(* IEC 61131-3 sources: open-ot-experiments/st/iec61131/src, 5 files *)

(* ---- openot_message.st ---- *)
FUNCTION_BLOCK OPENOT_EncodeMinimalMessage
VAR_INPUT
    SourceId : UDINT;
    RunId : ULINT;
    Seq : ULINT;
    SourceTime : ULINT;
    MessageTemplateId : UDINT;
END_VAR
VAR_OUTPUT
    Buffer : OPENOT_BYTE_BUFFER;
    Length : UINT;
END_VAR
VAR
    Pos : UINT;
    Crc : DWORD;
END_VAR

Pos := OPENOT_WriteHeader(
    TotalLength := UINT#52,
    Flags := UINT#16#0008,
    SourceTime := SourceTime,
    RunId := RunId,
    Seq := Seq,
    SourceId := SourceId,
    EventTypeId := UDINT#16#0003,
    Buffer := Buffer);

Pos := OPENOT_WriteSlotHeader(
    Offset := Pos,
    Key := UINT#16#0014,
    TypeTag := BYTE#16#05,
    PayloadLength := BYTE#4,
    Buffer := Buffer);
Pos := OPENOT_WriteU32LE(Offset := Pos, Value := MessageTemplateId, Buffer := Buffer);

Crc := OPENOT_Crc32c(Data := Buffer, Length := Pos);
Pos := OPENOT_WriteDWordLE(Offset := Pos, Value := Crc, Buffer := Buffer);
Length := Pos;
END_FUNCTION_BLOCK

(* ---- openot_producer.st ---- *)
TYPE
    OPENOT_SOURCE_ENTRY : STRUCT
        Used : BOOL;
        SourceId : UDINT;
        NextSeq : ULINT;
    END_STRUCT;

    OPENOT_SOURCE_USED_TABLE : ARRAY[0..15] OF BOOL;
    OPENOT_SOURCE_ID_TABLE : ARRAY[0..15] OF UDINT;
    OPENOT_SOURCE_NEXT_SEQ_TABLE : ARRAY[0..15] OF ULINT;
    OPENOT_SCAN_RECORD_BUFFER : ARRAY[0..1023] OF BYTE;
    OPENOT_SCAN_RECORD_UINT_TABLE : ARRAY[0..16] OF UINT;

    OPENOT_REAL_VALUE_STATE : STRUCT
        Used : BOOL;
        ValueId : UDINT;
        HasLast : BOOL;
        LastValue : REAL;
    END_STRUCT;

    OPENOT_INT_VALUE_STATE : STRUCT
        Used : BOOL;
        ValueId : UDINT;
        HasLast : BOOL;
        LastValue : DINT;
    END_STRUCT;

    OPENOT_STATE_MACHINE_STATE : STRUCT
        Used : BOOL;
        StateMachineId : UDINT;
        HasLast : BOOL;
        LastState : UINT;
    END_STRUCT;

    OPENOT_CONDITION_STATE : STRUCT
        Used : BOOL;
        ConditionId : UDINT;
        HasLast : BOOL;
        LastActive : BOOL;
    END_STRUCT;

    OPENOT_EMISSION_ENTRY : STRUCT
        EventTypeId : UDINT;
        RunId : ULINT;
        SourceId : UDINT;
        Seq : ULINT;
    END_STRUCT;

    OPENOT_EMISSION_LOG : ARRAY[0..31] OF OPENOT_EMISSION_ENTRY;
END_TYPE

FUNCTION OPENOT_AppendScanRecord : BOOL
VAR_INPUT
    Record : OPENOT_BYTE_BUFFER;
    Length : UINT;
END_VAR
VAR_IN_OUT
    ScanRecords : OPENOT_SCAN_RECORD_BUFFER;
    ScanRecordOffsets : OPENOT_SCAN_RECORD_UINT_TABLE;
    ScanRecordLengths : OPENOT_SCAN_RECORD_UINT_TABLE;
    ScanWritePos : UINT;
    ScanRecordCount : UINT;
END_VAR
VAR
    CopyIndex : UINT;
    DestIndex : UINT;
END_VAR

IF (Length = UINT#0) OR (Length > UINT#256) OR (ScanRecordCount > UINT#16) OR ((ScanWritePos + Length) > UINT#1024) THEN
    OPENOT_AppendScanRecord := FALSE;
ELSE
    ScanRecordOffsets[ScanRecordCount] := ScanWritePos;
    ScanRecordLengths[ScanRecordCount] := Length;

    FOR CopyIndex := UINT#0 TO Length - UINT#1 DO
        DestIndex := ScanWritePos + CopyIndex;
        ScanRecords[DestIndex] := Record[CopyIndex];
    END_FOR;

    ScanWritePos := ScanWritePos + Length;
    ScanRecordCount := ScanRecordCount + UINT#1;
    OPENOT_AppendScanRecord := TRUE;
END_IF;
END_FUNCTION

FUNCTION OPENOT_ResetScanRecordList : BOOL
VAR_IN_OUT
    ScanRecordOffsets : OPENOT_SCAN_RECORD_UINT_TABLE;
    ScanRecordLengths : OPENOT_SCAN_RECORD_UINT_TABLE;
    ScanWritePos : UINT;
    ScanRecordCount : UINT;
END_VAR
VAR
    Index : UINT;
END_VAR

ScanRecordCount := UINT#0;
ScanWritePos := UINT#0;
FOR Index := UINT#0 TO UINT#16 DO
    ScanRecordOffsets[Index] := UINT#0;
    ScanRecordLengths[Index] := UINT#0;
END_FOR;

OPENOT_ResetScanRecordList := TRUE;
END_FUNCTION

FUNCTION OPENOT_NextSourceTime : ULINT
VAR_INPUT
    UseSourceTimeInput : BOOL;
    SourceTimeInput : ULINT;
END_VAR
VAR_IN_OUT
    StateSourceTime : ULINT;
END_VAR

IF UseSourceTimeInput THEN
    OPENOT_NextSourceTime := SourceTimeInput;
ELSE
    OPENOT_NextSourceTime := StateSourceTime;
    StateSourceTime := StateSourceTime + ULINT#1;
END_IF;
END_FUNCTION

FUNCTION_BLOCK OPENOT_Producer
VAR_INPUT
    Execute : BOOL;
    Op : UINT;
    SourceId : UDINT;
    Checkpoint : BOOL;
    DefHashOld : OPENOT_HASH8;
    DefHashNew : OPENOT_HASH8;
    TransitionEpochId : ULINT;
    UseSourceTimeInput : BOOL;
    SourceTimeInput : ULINT;
    StageRecord : OPENOT_BYTE_BUFFER;
    StageLength : UINT;
    StageSeq : ULINT;
    StageEventTypeId : UDINT;
    ResetScanRecords : BOOL;
    AccumulateScanRecords : BOOL;
    ValueId : UDINT;
    ValueReal : REAL;
    ValueInt : DINT;
    DeadbandReal : REAL;
    HasQuality : BOOL;
    Quality : UINT;
    StateMachineId : UDINT;
    Category : UINT;
    PreviousState : UINT;
    NewState : UINT;
    ConditionId : UDINT;
    ConditionClass : UINT;
    Severity : UINT;
    ConditionActive : BOOL;
    MessageTemplateId : UDINT;
END_VAR
VAR_OUTPUT
    AssignedSeq : ULINT;
    ProducedCount : ULINT;
    Error : BOOL;
    SourceTableFull : BOOL;
    Done : BOOL;
    CheckpointDone : BOOL;
    SourceCount : UINT;
    SourceUsed : OPENOT_SOURCE_USED_TABLE;
    SourceIds : OPENOT_SOURCE_ID_TABLE;
    SourceNextSeqs : OPENOT_SOURCE_NEXT_SEQ_TABLE;
    Ring : OPENOT_RING256_BUFFER;
    HeadAbs : ULINT;
    OldestAbs : ULINT;
    LostCount : ULINT;
    LastStartAbs : ULINT;
    LastEndAbs : ULINT;
    LossRanges : OPENOT_PRODUCER_LOSS_RANGES;
    LossRangeCount : UINT;
    LossRangeOverflow : BOOL;
    RingError : BOOL;
    RunId : ULINT;
    SourceTime : ULINT;
    SystemSeq : ULINT;
    EpochId : ULINT;
    EpochFirstAbs : ULINT;
    DefinitionHash : OPENOT_HASH8;
    PrevDefinitionHash : OPENOT_HASH8;
    TransitionOpen : BOOL;
    DefinitionChangedEmitted : BOOL;
    Emissions : OPENOT_EMISSION_LOG;
    EmissionCount : UINT;
    PublishedRecordCount : ULINT;
    ScanRecords : OPENOT_SCAN_RECORD_BUFFER;
    ScanRecordOffsets : OPENOT_SCAN_RECORD_UINT_TABLE;
    ScanRecordLengths : OPENOT_SCAN_RECORD_UINT_TABLE;
    ScanRecordCount : UINT;
END_VAR
VAR
    Sources : ARRAY[0..15] OF OPENOT_SOURCE_ENTRY;
    RealValueStates : ARRAY[0..15] OF OPENOT_REAL_VALUE_STATE;
    IntValueStates : ARRAY[0..15] OF OPENOT_INT_VALUE_STATE;
    StateMachineStates : ARRAY[0..15] OF OPENOT_STATE_MACHINE_STATE;
    ConditionStates : ARRAY[0..15] OF OPENOT_CONDITION_STATE;
    RingProducer : OPENOT_Ring256Producer;
    Encoder : OPENOT_EncodeMinimalMessage;
    ValueRealEncoder : OPENOT_EncodeValueChangedReal;
    ValueIntEncoder : OPENOT_EncodeValueChangedInt;
    StateTransitionEncoder : OPENOT_EncodeStateTransition;
    ConditionEncoder : OPENOT_EncodeCondition;
    HighWaterEncoder : OPENOT_EncodeSourceHighWater;
    StoppedEncoder : OPENOT_EncodeLoggerStopped;
    StartedEncoder : OPENOT_EncodeLoggerStarted;
    DefinitionEncoder : OPENOT_EncodeDefinitionChanged;
    Index : UINT;
    ByteIndex : UINT;
    LossIndex : UINT;
    EntryIndex : UINT;
    Found : BOOL;
    FreeFound : BOOL;
    Initialized : BOOL;
    PreviousExecute : BOOL;
    ExecuteEdge : BOOL;
    StateRunId : ULINT;
    StateSourceTime : ULINT;
    StateSystemSeq : ULINT;
    StateEpochId : ULINT;
    StateEpochFirstAbs : ULINT;
    StateDefinitionHash : OPENOT_HASH8;
    StatePrevDefinitionHash : OPENOT_HASH8;
    StatePublishedRecordCount : ULINT;
    PendingDefHashOld : OPENOT_HASH8;
    PendingDefHashNew : OPENOT_HASH8;
    PendingEpochId : ULINT;
    PendingOpen : BOOL;
    PendingDefChangedEmitted : BOOL;
    EmitSeq : ULINT;
    EmitSourceTime : ULINT;
    SourceLoopActive : BOOL;
    HasLastSourceId : BOOL;
    LastSourceId : UDINT;
    NextSourceId : UDINT;
    SelectedIndex : UINT;
    StateIndex : UINT;
    StateFound : BOOL;
    StateFreeFound : BOOL;
    ActiveSourceId : UDINT;
    ShouldEmit : BOOL;
    DeltaReal : REAL;
    CandidateFound : BOOL;
    ScanWritePos : UINT;
    AppendOk : BOOL;
    ResetOk : BOOL;
    ConditionEventTypeId : UDINT;
END_VAR

IF NOT Initialized THEN
    StateRunId := ULINT#1;
    StateSourceTime := ULINT#1780000000000000000;
    StateSystemSeq := ULINT#0;
    StateEpochId := ULINT#1;
    StateEpochFirstAbs := ULINT#0;
    StatePublishedRecordCount := ULINT#0;
    Initialized := TRUE;
END_IF;

Done := FALSE;
Error := FALSE;
SourceTableFull := FALSE;
AssignedSeq := ULINT#0;
ProducedCount := ULINT#0;
CheckpointDone := FALSE;
ExecuteEdge := Execute AND (NOT PreviousExecute);

IF ResetScanRecords THEN
    ResetOk := OPENOT_ResetScanRecordList(
        ScanRecordOffsets := ScanRecordOffsets,
        ScanRecordLengths := ScanRecordLengths,
        ScanWritePos := ScanWritePos,
        ScanRecordCount := ScanRecordCount);
END_IF;

IF ExecuteEdge THEN
    IF (NOT AccumulateScanRecords) AND (Op <> UINT#6) AND (Op <> UINT#7) AND (Op <> UINT#8) AND (Op <> UINT#9) THEN
        ResetOk := OPENOT_ResetScanRecordList(
            ScanRecordOffsets := ScanRecordOffsets,
            ScanRecordLengths := ScanRecordLengths,
            ScanWritePos := ScanWritePos,
            ScanRecordCount := ScanRecordCount);
    END_IF;

    IF Checkpoint THEN
        IF PendingOpen THEN
            Error := TRUE;
        ELSIF SourceId = UDINT#0 THEN
            Error := TRUE;
        ELSE
            Found := FALSE;
            EntryIndex := UINT#0;

            FOR Index := UINT#0 TO UINT#15 DO
                IF Sources[Index].Used AND (Sources[Index].SourceId = SourceId) THEN
                    IF NOT Found THEN
                        EntryIndex := Index;
                        Found := TRUE;
                    END_IF;
                END_IF;
            END_FOR;

            IF NOT Found THEN
                Error := TRUE;
            ELSE
                ProducedCount := Sources[EntryIndex].NextSeq;
                EmitSourceTime := OPENOT_NextSourceTime(
                    UseSourceTimeInput := UseSourceTimeInput,
                    SourceTimeInput := SourceTimeInput,
                    StateSourceTime := StateSourceTime);
                HighWaterEncoder(
                    SourceId := SourceId,
                    RunId := StateRunId,
                    ProducedCount := ProducedCount,
                    SourceTime := EmitSourceTime);
                RingProducer(
                    Execute := TRUE,
                    Record := HighWaterEncoder.Buffer,
                    Length := HighWaterEncoder.Length,
                    RunId := StateRunId,
                    SourceId := SourceId,
                    Seq := ProducedCount);

                IF RingProducer.Done AND (NOT RingProducer.Error) THEN
                    AppendOk := OPENOT_AppendScanRecord(
                        Record := HighWaterEncoder.Buffer,
                        Length := HighWaterEncoder.Length,
                        ScanRecords := ScanRecords,
                        ScanRecordOffsets := ScanRecordOffsets,
                        ScanRecordLengths := ScanRecordLengths,
                        ScanWritePos := ScanWritePos,
                        ScanRecordCount := ScanRecordCount);
                    IF AppendOk THEN
                        Sources[EntryIndex].NextSeq := ProducedCount + ULINT#1;
                        StatePublishedRecordCount := StatePublishedRecordCount + ULINT#1;
                        IF EmissionCount < UINT#32 THEN
                            Emissions[EmissionCount].EventTypeId := UDINT#16#80000108;
                            Emissions[EmissionCount].RunId := StateRunId;
                            Emissions[EmissionCount].SourceId := SourceId;
                            Emissions[EmissionCount].Seq := ProducedCount;
                            EmissionCount := EmissionCount + UINT#1;
                        END_IF;
                        Done := TRUE;
                        CheckpointDone := TRUE;
                    ELSE
                        Error := TRUE;
                    END_IF;
                ELSE
                    Error := TRUE;
                END_IF;
            END_IF;
        END_IF;
    ELSIF Op = UINT#0 THEN
        IF PendingOpen THEN
            Error := TRUE;
        ELSIF SourceId = UDINT#0 THEN
            Error := TRUE;
        ELSE
            Found := FALSE;
            FreeFound := FALSE;
            EntryIndex := UINT#0;

            FOR Index := UINT#0 TO UINT#15 DO
                IF Sources[Index].Used AND (Sources[Index].SourceId = SourceId) THEN
                    IF NOT Found THEN
                        EntryIndex := Index;
                        Found := TRUE;
                    END_IF;
                END_IF;
            END_FOR;

            IF NOT Found THEN
                FOR Index := UINT#0 TO UINT#15 DO
                    IF (NOT Sources[Index].Used) AND (NOT FreeFound) THEN
                        EntryIndex := Index;
                        FreeFound := TRUE;
                    END_IF;
                END_FOR;

                IF FreeFound THEN
                    Sources[EntryIndex].Used := TRUE;
                    Sources[EntryIndex].SourceId := SourceId;
                    Sources[EntryIndex].NextSeq := ULINT#0;
                ELSE
                    SourceTableFull := TRUE;
                    Error := TRUE;
                END_IF;
            END_IF;

            IF NOT Error THEN
                AssignedSeq := Sources[EntryIndex].NextSeq;
                Sources[EntryIndex].NextSeq := Sources[EntryIndex].NextSeq + ULINT#1;
                EmitSourceTime := OPENOT_NextSourceTime(
                    UseSourceTimeInput := UseSourceTimeInput,
                    SourceTimeInput := SourceTimeInput,
                    StateSourceTime := StateSourceTime);

                Encoder(
                    SourceId := SourceId,
                    RunId := StateRunId,
                    Seq := AssignedSeq,
                    SourceTime := EmitSourceTime,
                    MessageTemplateId := MessageTemplateId);
                RingProducer(
                    Execute := TRUE,
                    Record := Encoder.Buffer,
                    Length := Encoder.Length,
                    RunId := StateRunId,
                    SourceId := SourceId,
                    Seq := AssignedSeq);

                IF RingProducer.Done AND (NOT RingProducer.Error) THEN
                    AppendOk := OPENOT_AppendScanRecord(
                        Record := Encoder.Buffer,
                        Length := Encoder.Length,
                        ScanRecords := ScanRecords,
                        ScanRecordOffsets := ScanRecordOffsets,
                        ScanRecordLengths := ScanRecordLengths,
                        ScanWritePos := ScanWritePos,
                        ScanRecordCount := ScanRecordCount);
                    IF AppendOk THEN
                        StatePublishedRecordCount := StatePublishedRecordCount + ULINT#1;
                        IF EmissionCount < UINT#32 THEN
                            Emissions[EmissionCount].EventTypeId := UDINT#16#0003;
                            Emissions[EmissionCount].RunId := StateRunId;
                            Emissions[EmissionCount].SourceId := SourceId;
                            Emissions[EmissionCount].Seq := AssignedSeq;
                            EmissionCount := EmissionCount + UINT#1;
                        END_IF;
                        Done := TRUE;
                    ELSE
                        Error := TRUE;
                    END_IF;
                ELSE
                    Error := TRUE;
                END_IF;
            END_IF;
        END_IF;
    ELSIF Op = UINT#5 THEN
        IF PendingOpen THEN
            Error := TRUE;
        ELSIF SourceId = UDINT#0 THEN
            Error := TRUE;
        ELSIF (StageLength = UINT#0) OR (StageLength > UINT#256) THEN
            Error := TRUE;
        ELSE
            Found := FALSE;
            FreeFound := FALSE;
            EntryIndex := UINT#0;

            FOR Index := UINT#0 TO UINT#15 DO
                IF Sources[Index].Used AND (Sources[Index].SourceId = SourceId) THEN
                    IF NOT Found THEN
                        EntryIndex := Index;
                        Found := TRUE;
                    END_IF;
                END_IF;
            END_FOR;

            IF NOT Found THEN
                FOR Index := UINT#0 TO UINT#15 DO
                    IF (NOT Sources[Index].Used) AND (NOT FreeFound) THEN
                        EntryIndex := Index;
                        FreeFound := TRUE;
                    END_IF;
                END_FOR;

                IF FreeFound THEN
                    Sources[EntryIndex].Used := TRUE;
                    Sources[EntryIndex].SourceId := SourceId;
                    Sources[EntryIndex].NextSeq := ULINT#0;
                ELSE
                    SourceTableFull := TRUE;
                    Error := TRUE;
                END_IF;
            END_IF;

            IF NOT Error THEN
                IF StageSeq <> Sources[EntryIndex].NextSeq THEN
                    Error := TRUE;
                ELSE
                    RingProducer(
                        Execute := TRUE,
                        Record := StageRecord,
                        Length := StageLength,
                        RunId := StateRunId,
                        SourceId := SourceId,
                        Seq := StageSeq);

                    IF RingProducer.Done AND (NOT RingProducer.Error) THEN
                        AppendOk := OPENOT_AppendScanRecord(
                            Record := StageRecord,
                            Length := StageLength,
                            ScanRecords := ScanRecords,
                            ScanRecordOffsets := ScanRecordOffsets,
                            ScanRecordLengths := ScanRecordLengths,
                            ScanWritePos := ScanWritePos,
                            ScanRecordCount := ScanRecordCount);
                        IF AppendOk THEN
                            AssignedSeq := StageSeq;
                            Sources[EntryIndex].NextSeq := StageSeq + ULINT#1;
                            StatePublishedRecordCount := StatePublishedRecordCount + ULINT#1;
                            IF EmissionCount < UINT#32 THEN
                                Emissions[EmissionCount].EventTypeId := StageEventTypeId;
                                Emissions[EmissionCount].RunId := StateRunId;
                                Emissions[EmissionCount].SourceId := SourceId;
                                Emissions[EmissionCount].Seq := StageSeq;
                                EmissionCount := EmissionCount + UINT#1;
                            END_IF;
                            Done := TRUE;
                        ELSE
                            Error := TRUE;
                        END_IF;
                    ELSE
                        Error := TRUE;
                    END_IF;
                END_IF;
            END_IF;
        END_IF;
    ELSIF (Op = UINT#6) OR (Op = UINT#7) OR (Op = UINT#8) THEN
        ActiveSourceId := SourceId;
        IF ActiveSourceId = UDINT#0 THEN
            ActiveSourceId := UDINT#1;
        END_IF;

        StateFound := FALSE;
        StateFreeFound := FALSE;
        StateIndex := UINT#0;
        ShouldEmit := FALSE;

        IF Op = UINT#6 THEN
            IF ValueId = UDINT#0 THEN
                Error := TRUE;
            ELSE
                FOR Index := UINT#0 TO UINT#15 DO
                    IF RealValueStates[Index].Used AND (RealValueStates[Index].ValueId = ValueId) THEN
                        IF NOT StateFound THEN
                            StateIndex := Index;
                            StateFound := TRUE;
                        END_IF;
                    ELSIF (NOT StateFound) AND (NOT RealValueStates[Index].Used) AND (NOT StateFreeFound) THEN
                        StateIndex := Index;
                        StateFreeFound := TRUE;
                    END_IF;
                END_FOR;

                IF StateFound THEN
                    IF RealValueStates[StateIndex].HasLast THEN
                        DeltaReal := ValueReal - RealValueStates[StateIndex].LastValue;
                        IF DeltaReal < REAL#0.0 THEN
                            DeltaReal := REAL#0.0 - DeltaReal;
                        END_IF;
                        ShouldEmit := DeltaReal > DeadbandReal;
                    ELSE
                        ShouldEmit := TRUE;
                    END_IF;
                ELSIF StateFreeFound THEN
                    RealValueStates[StateIndex].Used := TRUE;
                    RealValueStates[StateIndex].ValueId := ValueId;
                    RealValueStates[StateIndex].HasLast := FALSE;
                    ShouldEmit := TRUE;
                ELSE
                    Error := TRUE;
                END_IF;
            END_IF;
        ELSIF Op = UINT#7 THEN
            IF ValueId = UDINT#0 THEN
                Error := TRUE;
            ELSE
                FOR Index := UINT#0 TO UINT#15 DO
                    IF IntValueStates[Index].Used AND (IntValueStates[Index].ValueId = ValueId) THEN
                        IF NOT StateFound THEN
                            StateIndex := Index;
                            StateFound := TRUE;
                        END_IF;
                    ELSIF (NOT StateFound) AND (NOT IntValueStates[Index].Used) AND (NOT StateFreeFound) THEN
                        StateIndex := Index;
                        StateFreeFound := TRUE;
                    END_IF;
                END_FOR;

                IF StateFound THEN
                    IF IntValueStates[StateIndex].HasLast THEN
                        ShouldEmit := ValueInt <> IntValueStates[StateIndex].LastValue;
                    ELSE
                        ShouldEmit := TRUE;
                    END_IF;
                ELSIF StateFreeFound THEN
                    IntValueStates[StateIndex].Used := TRUE;
                    IntValueStates[StateIndex].ValueId := ValueId;
                    IntValueStates[StateIndex].HasLast := FALSE;
                    ShouldEmit := TRUE;
                ELSE
                    Error := TRUE;
                END_IF;
            END_IF;
        ELSE
            IF StateMachineId = UDINT#0 THEN
                Error := TRUE;
            ELSE
                FOR Index := UINT#0 TO UINT#15 DO
                    IF StateMachineStates[Index].Used AND (StateMachineStates[Index].StateMachineId = StateMachineId) THEN
                        IF NOT StateFound THEN
                            StateIndex := Index;
                            StateFound := TRUE;
                        END_IF;
                    ELSIF (NOT StateFound) AND (NOT StateMachineStates[Index].Used) AND (NOT StateFreeFound) THEN
                        StateIndex := Index;
                        StateFreeFound := TRUE;
                    END_IF;
                END_FOR;

                IF PreviousState <> NewState THEN
                    IF StateFound THEN
                        ShouldEmit := (NOT StateMachineStates[StateIndex].HasLast) OR (StateMachineStates[StateIndex].LastState <> NewState);
                    ELSIF StateFreeFound THEN
                        StateMachineStates[StateIndex].Used := TRUE;
                        StateMachineStates[StateIndex].StateMachineId := StateMachineId;
                        StateMachineStates[StateIndex].HasLast := FALSE;
                        ShouldEmit := TRUE;
                    ELSE
                        Error := TRUE;
                    END_IF;
                ELSE
                    ShouldEmit := FALSE;
                END_IF;
            END_IF;
        END_IF;

        IF (NOT Error) AND (NOT ShouldEmit) THEN
            Done := TRUE;
        ELSIF NOT Error THEN
            Found := FALSE;
            FreeFound := FALSE;
            EntryIndex := UINT#0;

            FOR Index := UINT#0 TO UINT#15 DO
                IF Sources[Index].Used AND (Sources[Index].SourceId = ActiveSourceId) THEN
                    IF NOT Found THEN
                        EntryIndex := Index;
                        Found := TRUE;
                    END_IF;
                END_IF;
            END_FOR;

            IF NOT Found THEN
                FOR Index := UINT#0 TO UINT#15 DO
                    IF (NOT Sources[Index].Used) AND (NOT FreeFound) THEN
                        EntryIndex := Index;
                        FreeFound := TRUE;
                    END_IF;
                END_FOR;

                IF FreeFound THEN
                    Sources[EntryIndex].Used := TRUE;
                    Sources[EntryIndex].SourceId := ActiveSourceId;
                    Sources[EntryIndex].NextSeq := ULINT#0;
                ELSE
                    SourceTableFull := TRUE;
                    Error := TRUE;
                END_IF;
            END_IF;

            IF NOT Error THEN
                AssignedSeq := Sources[EntryIndex].NextSeq;
                EmitSourceTime := OPENOT_NextSourceTime(
                    UseSourceTimeInput := UseSourceTimeInput,
                    SourceTimeInput := SourceTimeInput,
                    StateSourceTime := StateSourceTime);

                IF Op = UINT#6 THEN
                    ValueRealEncoder(
                        SourceId := ActiveSourceId,
                        RunId := StateRunId,
                        Seq := AssignedSeq,
                        SourceTime := EmitSourceTime,
                        ValueId := ValueId,
                        NewValue := ValueReal,
                        HasPrevious := RealValueStates[StateIndex].HasLast,
                        PreviousValue := RealValueStates[StateIndex].LastValue,
                        HasQuality := HasQuality,
                        Quality := Quality);
                    RingProducer(
                        Execute := TRUE,
                        Record := ValueRealEncoder.Buffer,
                        Length := ValueRealEncoder.Length,
                        RunId := StateRunId,
                        SourceId := ActiveSourceId,
                        Seq := AssignedSeq);

                    IF RingProducer.Done AND (NOT RingProducer.Error) THEN
                        AppendOk := OPENOT_AppendScanRecord(
                            Record := ValueRealEncoder.Buffer,
                            Length := ValueRealEncoder.Length,
                            ScanRecords := ScanRecords,
                            ScanRecordOffsets := ScanRecordOffsets,
                            ScanRecordLengths := ScanRecordLengths,
                            ScanWritePos := ScanWritePos,
                            ScanRecordCount := ScanRecordCount);
                    ELSE
                        AppendOk := FALSE;
                    END_IF;
                ELSIF Op = UINT#7 THEN
                    ValueIntEncoder(
                        SourceId := ActiveSourceId,
                        RunId := StateRunId,
                        Seq := AssignedSeq,
                        SourceTime := EmitSourceTime,
                        ValueId := ValueId,
                        NewValue := ValueInt,
                        HasPrevious := IntValueStates[StateIndex].HasLast,
                        PreviousValue := IntValueStates[StateIndex].LastValue,
                        HasQuality := HasQuality,
                        Quality := Quality);
                    RingProducer(
                        Execute := TRUE,
                        Record := ValueIntEncoder.Buffer,
                        Length := ValueIntEncoder.Length,
                        RunId := StateRunId,
                        SourceId := ActiveSourceId,
                        Seq := AssignedSeq);

                    IF RingProducer.Done AND (NOT RingProducer.Error) THEN
                        AppendOk := OPENOT_AppendScanRecord(
                            Record := ValueIntEncoder.Buffer,
                            Length := ValueIntEncoder.Length,
                            ScanRecords := ScanRecords,
                            ScanRecordOffsets := ScanRecordOffsets,
                            ScanRecordLengths := ScanRecordLengths,
                            ScanWritePos := ScanWritePos,
                            ScanRecordCount := ScanRecordCount);
                    ELSE
                        AppendOk := FALSE;
                    END_IF;
                ELSE
                    StateTransitionEncoder(
                        SourceId := ActiveSourceId,
                        RunId := StateRunId,
                        Seq := AssignedSeq,
                        SourceTime := EmitSourceTime,
                        StateMachineId := StateMachineId,
                        Category := Category,
                        PreviousState := PreviousState,
                        NewState := NewState);
                    RingProducer(
                        Execute := TRUE,
                        Record := StateTransitionEncoder.Buffer,
                        Length := StateTransitionEncoder.Length,
                        RunId := StateRunId,
                        SourceId := ActiveSourceId,
                        Seq := AssignedSeq);

                    IF RingProducer.Done AND (NOT RingProducer.Error) THEN
                        AppendOk := OPENOT_AppendScanRecord(
                            Record := StateTransitionEncoder.Buffer,
                            Length := StateTransitionEncoder.Length,
                            ScanRecords := ScanRecords,
                            ScanRecordOffsets := ScanRecordOffsets,
                            ScanRecordLengths := ScanRecordLengths,
                            ScanWritePos := ScanWritePos,
                            ScanRecordCount := ScanRecordCount);
                    ELSE
                        AppendOk := FALSE;
                    END_IF;
                END_IF;

                IF AppendOk THEN
                    Sources[EntryIndex].NextSeq := AssignedSeq + ULINT#1;
                    StatePublishedRecordCount := StatePublishedRecordCount + ULINT#1;
                    IF EmissionCount < UINT#32 THEN
                        IF Op = UINT#8 THEN
                            Emissions[EmissionCount].EventTypeId := UDINT#16#0001;
                        ELSE
                            Emissions[EmissionCount].EventTypeId := UDINT#16#0002;
                        END_IF;
                        Emissions[EmissionCount].RunId := StateRunId;
                        Emissions[EmissionCount].SourceId := ActiveSourceId;
                        Emissions[EmissionCount].Seq := AssignedSeq;
                        EmissionCount := EmissionCount + UINT#1;
                    END_IF;

                    IF Op = UINT#6 THEN
                        RealValueStates[StateIndex].HasLast := TRUE;
                        RealValueStates[StateIndex].LastValue := ValueReal;
                    ELSIF Op = UINT#7 THEN
                        IntValueStates[StateIndex].HasLast := TRUE;
                        IntValueStates[StateIndex].LastValue := ValueInt;
                    ELSE
                        StateMachineStates[StateIndex].HasLast := TRUE;
                        StateMachineStates[StateIndex].LastState := NewState;
                    END_IF;
                    Done := TRUE;
                ELSE
                    Error := TRUE;
                END_IF;
            END_IF;
        END_IF;
    ELSIF Op = UINT#9 THEN
        ActiveSourceId := SourceId;
        IF ActiveSourceId = UDINT#0 THEN
            ActiveSourceId := UDINT#1;
        END_IF;

        StateFound := FALSE;
        StateFreeFound := FALSE;
        StateIndex := UINT#0;
        ShouldEmit := FALSE;

        IF ConditionId = UDINT#0 THEN
            Error := TRUE;
        ELSE
            FOR Index := UINT#0 TO UINT#15 DO
                IF ConditionStates[Index].Used AND (ConditionStates[Index].ConditionId = ConditionId) THEN
                    IF NOT StateFound THEN
                        StateIndex := Index;
                        StateFound := TRUE;
                    END_IF;
                ELSIF (NOT StateFound) AND (NOT ConditionStates[Index].Used) AND (NOT StateFreeFound) THEN
                    StateIndex := Index;
                    StateFreeFound := TRUE;
                END_IF;
            END_FOR;

            IF StateFound THEN
                IF ConditionStates[StateIndex].HasLast THEN
                    ShouldEmit := ConditionStates[StateIndex].LastActive <> ConditionActive;
                ELSE
                    ShouldEmit := ConditionActive;
                END_IF;
            ELSIF StateFreeFound THEN
                ConditionStates[StateIndex].Used := TRUE;
                ConditionStates[StateIndex].ConditionId := ConditionId;
                ConditionStates[StateIndex].HasLast := FALSE;
                ShouldEmit := ConditionActive;
            ELSE
                Error := TRUE;
            END_IF;
        END_IF;

        IF (NOT Error) AND (NOT ShouldEmit) THEN
            IF StateFound OR StateFreeFound THEN
                ConditionStates[StateIndex].HasLast := TRUE;
                ConditionStates[StateIndex].LastActive := ConditionActive;
            END_IF;
            Done := TRUE;
        ELSIF NOT Error THEN
            Found := FALSE;
            FreeFound := FALSE;
            EntryIndex := UINT#0;

            FOR Index := UINT#0 TO UINT#15 DO
                IF Sources[Index].Used AND (Sources[Index].SourceId = ActiveSourceId) THEN
                    IF NOT Found THEN
                        EntryIndex := Index;
                        Found := TRUE;
                    END_IF;
                END_IF;
            END_FOR;

            IF NOT Found THEN
                FOR Index := UINT#0 TO UINT#15 DO
                    IF (NOT Sources[Index].Used) AND (NOT FreeFound) THEN
                        EntryIndex := Index;
                        FreeFound := TRUE;
                    END_IF;
                END_FOR;

                IF FreeFound THEN
                    Sources[EntryIndex].Used := TRUE;
                    Sources[EntryIndex].SourceId := ActiveSourceId;
                    Sources[EntryIndex].NextSeq := ULINT#0;
                ELSE
                    SourceTableFull := TRUE;
                    Error := TRUE;
                END_IF;
            END_IF;

            IF NOT Error THEN
                AssignedSeq := Sources[EntryIndex].NextSeq;
                EmitSourceTime := OPENOT_NextSourceTime(
                    UseSourceTimeInput := UseSourceTimeInput,
                    SourceTimeInput := SourceTimeInput,
                    StateSourceTime := StateSourceTime);
                IF ConditionActive THEN
                    ConditionEventTypeId := UDINT#16#0200;
                ELSE
                    ConditionEventTypeId := UDINT#16#0201;
                END_IF;

                ConditionEncoder(
                    SourceId := ActiveSourceId,
                    RunId := StateRunId,
                    Seq := AssignedSeq,
                    SourceTime := EmitSourceTime,
                    EventTypeId := ConditionEventTypeId,
                    ConditionId := ConditionId,
                    ConditionClass := ConditionClass,
                    Severity := Severity);
                RingProducer(
                    Execute := TRUE,
                    Record := ConditionEncoder.Buffer,
                    Length := ConditionEncoder.Length,
                    RunId := StateRunId,
                    SourceId := ActiveSourceId,
                    Seq := AssignedSeq);

                IF RingProducer.Done AND (NOT RingProducer.Error) THEN
                    AppendOk := OPENOT_AppendScanRecord(
                        Record := ConditionEncoder.Buffer,
                        Length := ConditionEncoder.Length,
                        ScanRecords := ScanRecords,
                        ScanRecordOffsets := ScanRecordOffsets,
                        ScanRecordLengths := ScanRecordLengths,
                        ScanWritePos := ScanWritePos,
                        ScanRecordCount := ScanRecordCount);
                ELSE
                    AppendOk := FALSE;
                END_IF;

                IF AppendOk THEN
                    Sources[EntryIndex].NextSeq := AssignedSeq + ULINT#1;
                    StatePublishedRecordCount := StatePublishedRecordCount + ULINT#1;
                    IF EmissionCount < UINT#32 THEN
                        Emissions[EmissionCount].EventTypeId := ConditionEventTypeId;
                        Emissions[EmissionCount].RunId := StateRunId;
                        Emissions[EmissionCount].SourceId := ActiveSourceId;
                        Emissions[EmissionCount].Seq := AssignedSeq;
                        EmissionCount := EmissionCount + UINT#1;
                    END_IF;
                    ConditionStates[StateIndex].HasLast := TRUE;
                    ConditionStates[StateIndex].LastActive := ConditionActive;
                    Done := TRUE;
                ELSE
                    Error := TRUE;
                END_IF;
            END_IF;
        END_IF;
    ELSIF Op = UINT#1 THEN
        IF PendingOpen THEN
            Error := TRUE;
        ELSE
            EmitSeq := StateSystemSeq;
            StateSystemSeq := StateSystemSeq + ULINT#1;
            EmitSourceTime := OPENOT_NextSourceTime(
                UseSourceTimeInput := UseSourceTimeInput,
                SourceTimeInput := SourceTimeInput,
                StateSourceTime := StateSourceTime);
            StoppedEncoder(RunId := StateRunId, Seq := EmitSeq, SourceTime := EmitSourceTime);
            RingProducer(
                Execute := TRUE,
                Record := StoppedEncoder.Buffer,
                Length := StoppedEncoder.Length,
                RunId := StateRunId,
                SourceId := UDINT#0,
                Seq := EmitSeq);

            IF RingProducer.Done AND (NOT RingProducer.Error) THEN
                AppendOk := OPENOT_AppendScanRecord(
                    Record := StoppedEncoder.Buffer,
                    Length := StoppedEncoder.Length,
                    ScanRecords := ScanRecords,
                    ScanRecordOffsets := ScanRecordOffsets,
                    ScanRecordLengths := ScanRecordLengths,
                    ScanWritePos := ScanWritePos,
                    ScanRecordCount := ScanRecordCount);
                IF AppendOk THEN
                    StatePublishedRecordCount := StatePublishedRecordCount + ULINT#1;
                    IF EmissionCount < UINT#32 THEN
                        Emissions[EmissionCount].EventTypeId := UDINT#16#0102;
                        Emissions[EmissionCount].RunId := StateRunId;
                        Emissions[EmissionCount].SourceId := UDINT#0;
                        Emissions[EmissionCount].Seq := EmitSeq;
                        EmissionCount := EmissionCount + UINT#1;
                    END_IF;
                ELSE
                    Error := TRUE;
                END_IF;
            ELSE
                Error := TRUE;
            END_IF;

            SourceLoopActive := NOT Error;
            HasLastSourceId := FALSE;
            LastSourceId := UDINT#0;

            WHILE SourceLoopActive DO
                CandidateFound := FALSE;
                SelectedIndex := UINT#0;
                NextSourceId := UDINT#0;

                FOR Index := UINT#0 TO UINT#15 DO
                    IF Sources[Index].Used AND ((NOT HasLastSourceId) OR (Sources[Index].SourceId > LastSourceId)) THEN
                        IF (NOT CandidateFound) OR (Sources[Index].SourceId < NextSourceId) THEN
                            CandidateFound := TRUE;
                            SelectedIndex := Index;
                            NextSourceId := Sources[Index].SourceId;
                        END_IF;
                    END_IF;
                END_FOR;

                IF CandidateFound THEN
                    ProducedCount := Sources[SelectedIndex].NextSeq;
                    EmitSourceTime := OPENOT_NextSourceTime(
                        UseSourceTimeInput := UseSourceTimeInput,
                        SourceTimeInput := SourceTimeInput,
                        StateSourceTime := StateSourceTime);
                    HighWaterEncoder(
                        SourceId := Sources[SelectedIndex].SourceId,
                        RunId := StateRunId,
                        ProducedCount := ProducedCount,
                        SourceTime := EmitSourceTime);
                    RingProducer(
                        Execute := TRUE,
                        Record := HighWaterEncoder.Buffer,
                        Length := HighWaterEncoder.Length,
                        RunId := StateRunId,
                        SourceId := Sources[SelectedIndex].SourceId,
                        Seq := ProducedCount);

                    IF RingProducer.Done AND (NOT RingProducer.Error) THEN
                        AppendOk := OPENOT_AppendScanRecord(
                            Record := HighWaterEncoder.Buffer,
                            Length := HighWaterEncoder.Length,
                            ScanRecords := ScanRecords,
                            ScanRecordOffsets := ScanRecordOffsets,
                            ScanRecordLengths := ScanRecordLengths,
                            ScanWritePos := ScanWritePos,
                            ScanRecordCount := ScanRecordCount);
                        IF AppendOk THEN
                            Sources[SelectedIndex].NextSeq := ProducedCount + ULINT#1;
                            StatePublishedRecordCount := StatePublishedRecordCount + ULINT#1;
                            IF EmissionCount < UINT#32 THEN
                                Emissions[EmissionCount].EventTypeId := UDINT#16#80000108;
                                Emissions[EmissionCount].RunId := StateRunId;
                                Emissions[EmissionCount].SourceId := Sources[SelectedIndex].SourceId;
                                Emissions[EmissionCount].Seq := ProducedCount;
                                EmissionCount := EmissionCount + UINT#1;
                            END_IF;
                            LastSourceId := NextSourceId;
                            HasLastSourceId := TRUE;
                        ELSE
                            Error := TRUE;
                            SourceLoopActive := FALSE;
                        END_IF;
                    ELSE
                        Error := TRUE;
                        SourceLoopActive := FALSE;
                    END_IF;
                ELSE
                    SourceLoopActive := FALSE;
                END_IF;
            END_WHILE;

            IF NOT Error THEN
                FOR Index := UINT#0 TO UINT#7 DO
                    PendingDefHashOld[Index] := DefHashOld[Index];
                    PendingDefHashNew[Index] := DefHashNew[Index];
                END_FOR;
                PendingEpochId := TransitionEpochId;
                PendingDefChangedEmitted := FALSE;
                PendingOpen := TRUE;
                Done := TRUE;
            END_IF;
        END_IF;
    ELSIF Op = UINT#2 THEN
        IF NOT PendingOpen THEN
            Error := TRUE;
        ELSIF PendingDefChangedEmitted THEN
            Error := TRUE;
        ELSE
            EmitSeq := StateSystemSeq;
            StateSystemSeq := StateSystemSeq + ULINT#1;
            EmitSourceTime := OPENOT_NextSourceTime(
                UseSourceTimeInput := UseSourceTimeInput,
                SourceTimeInput := SourceTimeInput,
                StateSourceTime := StateSourceTime);
            DefinitionEncoder(
                RunId := StateRunId,
                Seq := EmitSeq,
                DefHashOld := PendingDefHashOld,
                DefHashNew := PendingDefHashNew,
                EpochId := PendingEpochId,
                SourceTime := EmitSourceTime);
            RingProducer(
                Execute := TRUE,
                Record := DefinitionEncoder.Buffer,
                Length := DefinitionEncoder.Length,
                RunId := StateRunId,
                SourceId := UDINT#0,
                Seq := EmitSeq);

            IF RingProducer.Done AND (NOT RingProducer.Error) THEN
                AppendOk := OPENOT_AppendScanRecord(
                    Record := DefinitionEncoder.Buffer,
                    Length := DefinitionEncoder.Length,
                    ScanRecords := ScanRecords,
                    ScanRecordOffsets := ScanRecordOffsets,
                    ScanRecordLengths := ScanRecordLengths,
                    ScanWritePos := ScanWritePos,
                    ScanRecordCount := ScanRecordCount);
                IF AppendOk THEN
                    StatePublishedRecordCount := StatePublishedRecordCount + ULINT#1;
                    IF EmissionCount < UINT#32 THEN
                        Emissions[EmissionCount].EventTypeId := UDINT#16#0106;
                        Emissions[EmissionCount].RunId := StateRunId;
                        Emissions[EmissionCount].SourceId := UDINT#0;
                        Emissions[EmissionCount].Seq := EmitSeq;
                        EmissionCount := EmissionCount + UINT#1;
                    END_IF;
                    PendingDefChangedEmitted := TRUE;
                    Done := TRUE;
                ELSE
                    Error := TRUE;
                END_IF;
            ELSE
                Error := TRUE;
            END_IF;
        END_IF;
    ELSIF Op = UINT#3 THEN
        IF NOT PendingOpen THEN
            Error := TRUE;
        ELSIF NOT PendingDefChangedEmitted THEN
            Error := TRUE;
        ELSE
            StateEpochId := PendingEpochId;
            EmitSeq := StateSystemSeq;
            StateSystemSeq := StateSystemSeq + ULINT#1;
            EmitSourceTime := OPENOT_NextSourceTime(
                UseSourceTimeInput := UseSourceTimeInput,
                SourceTimeInput := SourceTimeInput,
                StateSourceTime := StateSourceTime);
            StartedEncoder(
                RunId := StateRunId,
                Seq := EmitSeq,
                ColdStart := FALSE,
                SourceTime := EmitSourceTime);
            RingProducer(
                Execute := TRUE,
                Record := StartedEncoder.Buffer,
                Length := StartedEncoder.Length,
                RunId := StateRunId,
                SourceId := UDINT#0,
                Seq := EmitSeq);

            IF RingProducer.Done AND (NOT RingProducer.Error) THEN
                AppendOk := OPENOT_AppendScanRecord(
                    Record := StartedEncoder.Buffer,
                    Length := StartedEncoder.Length,
                    ScanRecords := ScanRecords,
                    ScanRecordOffsets := ScanRecordOffsets,
                    ScanRecordLengths := ScanRecordLengths,
                    ScanWritePos := ScanWritePos,
                    ScanRecordCount := ScanRecordCount);
                IF AppendOk THEN
                    StateEpochFirstAbs := RingProducer.LastStartAbs;
                    FOR Index := UINT#0 TO UINT#7 DO
                        StatePrevDefinitionHash[Index] := PendingDefHashOld[Index];
                        StateDefinitionHash[Index] := PendingDefHashNew[Index];
                    END_FOR;
                    PendingOpen := FALSE;
                    PendingDefChangedEmitted := FALSE;
                    StatePublishedRecordCount := StatePublishedRecordCount + ULINT#1;
                    IF EmissionCount < UINT#32 THEN
                        Emissions[EmissionCount].EventTypeId := UDINT#16#0101;
                        Emissions[EmissionCount].RunId := StateRunId;
                        Emissions[EmissionCount].SourceId := UDINT#0;
                        Emissions[EmissionCount].Seq := EmitSeq;
                        EmissionCount := EmissionCount + UINT#1;
                    END_IF;
                    Done := TRUE;
                ELSE
                    Error := TRUE;
                END_IF;
            ELSE
                Error := TRUE;
            END_IF;
        END_IF;
    ELSIF Op = UINT#4 THEN
        IF NOT PendingOpen THEN
            Error := TRUE;
        ELSIF NOT PendingDefChangedEmitted THEN
            Error := TRUE;
        ELSE
            StateRunId := StateRunId + ULINT#1;
            StateEpochId := PendingEpochId;
            StateSystemSeq := ULINT#0;

            FOR Index := UINT#0 TO UINT#15 DO
                Sources[Index].Used := FALSE;
                Sources[Index].SourceId := UDINT#0;
                Sources[Index].NextSeq := ULINT#0;
            END_FOR;

            EmitSeq := StateSystemSeq;
            StateSystemSeq := StateSystemSeq + ULINT#1;
            EmitSourceTime := OPENOT_NextSourceTime(
                UseSourceTimeInput := UseSourceTimeInput,
                SourceTimeInput := SourceTimeInput,
                StateSourceTime := StateSourceTime);
            StartedEncoder(
                RunId := StateRunId,
                Seq := EmitSeq,
                ColdStart := TRUE,
                SourceTime := EmitSourceTime);
            RingProducer(
                Execute := TRUE,
                Record := StartedEncoder.Buffer,
                Length := StartedEncoder.Length,
                RunId := StateRunId,
                SourceId := UDINT#0,
                Seq := EmitSeq);

            IF RingProducer.Done AND (NOT RingProducer.Error) THEN
                AppendOk := OPENOT_AppendScanRecord(
                    Record := StartedEncoder.Buffer,
                    Length := StartedEncoder.Length,
                    ScanRecords := ScanRecords,
                    ScanRecordOffsets := ScanRecordOffsets,
                    ScanRecordLengths := ScanRecordLengths,
                    ScanWritePos := ScanWritePos,
                    ScanRecordCount := ScanRecordCount);
                IF AppendOk THEN
                    StateEpochFirstAbs := RingProducer.LastStartAbs;
                    FOR Index := UINT#0 TO UINT#7 DO
                        StatePrevDefinitionHash[Index] := PendingDefHashOld[Index];
                        StateDefinitionHash[Index] := PendingDefHashNew[Index];
                    END_FOR;
                    PendingOpen := FALSE;
                    PendingDefChangedEmitted := FALSE;
                    StatePublishedRecordCount := StatePublishedRecordCount + ULINT#1;
                    IF EmissionCount < UINT#32 THEN
                        Emissions[EmissionCount].EventTypeId := UDINT#16#0101;
                        Emissions[EmissionCount].RunId := StateRunId;
                        Emissions[EmissionCount].SourceId := UDINT#0;
                        Emissions[EmissionCount].Seq := EmitSeq;
                        EmissionCount := EmissionCount + UINT#1;
                    END_IF;
                    Done := TRUE;
                ELSE
                    Error := TRUE;
                END_IF;
            ELSE
                Error := TRUE;
            END_IF;
        END_IF;
    ELSE
        Error := TRUE;
    END_IF;
END_IF;

PreviousExecute := Execute;

SourceCount := UINT#0;
FOR Index := UINT#0 TO UINT#15 DO
    SourceUsed[Index] := Sources[Index].Used;
    SourceIds[Index] := Sources[Index].SourceId;
    SourceNextSeqs[Index] := Sources[Index].NextSeq;
    IF Sources[Index].Used THEN
        SourceCount := SourceCount + UINT#1;
    END_IF;
END_FOR;

RunId := StateRunId;
IF UseSourceTimeInput THEN
    SourceTime := SourceTimeInput;
ELSE
    SourceTime := StateSourceTime;
END_IF;
SystemSeq := StateSystemSeq;
PublishedRecordCount := StatePublishedRecordCount;
EpochId := StateEpochId;
EpochFirstAbs := StateEpochFirstAbs;
TransitionOpen := PendingOpen;
DefinitionChangedEmitted := PendingDefChangedEmitted;

FOR Index := UINT#0 TO UINT#7 DO
    DefinitionHash[Index] := StateDefinitionHash[Index];
    PrevDefinitionHash[Index] := StatePrevDefinitionHash[Index];
END_FOR;

IF ExecuteEdge THEN
    FOR ByteIndex := UINT#0 TO UINT#255 DO
        Ring[ByteIndex] := RingProducer.Ring[ByteIndex];
    END_FOR;

    FOR LossIndex := UINT#0 TO UINT#15 DO
        LossRanges[LossIndex].RunId := RingProducer.LossRanges[LossIndex].RunId;
        LossRanges[LossIndex].SourceId := RingProducer.LossRanges[LossIndex].SourceId;
        LossRanges[LossIndex].FirstSeq := RingProducer.LossRanges[LossIndex].FirstSeq;
        LossRanges[LossIndex].LastSeq := RingProducer.LossRanges[LossIndex].LastSeq;
    END_FOR;

    HeadAbs := RingProducer.HeadAbs;
    OldestAbs := RingProducer.OldestAbs;
    LostCount := RingProducer.LostCount;
    LastStartAbs := RingProducer.LastStartAbs;
    LastEndAbs := RingProducer.LastEndAbs;
    LossRangeCount := RingProducer.LossRangeCount;
    LossRangeOverflow := RingProducer.LossRangeOverflow;
    RingError := RingProducer.Error;
END_IF;
END_FUNCTION_BLOCK

(* ---- openot_source_high_water.st ---- *)
FUNCTION_BLOCK OPENOT_EncodeSourceHighWater
VAR_INPUT
    SourceId : UDINT;
    RunId : ULINT;
    ProducedCount : ULINT;
    SourceTime : ULINT;
END_VAR
VAR_OUTPUT
    Buffer : OPENOT_BYTE_BUFFER;
    Length : UINT;
END_VAR
VAR
    Pos : UINT;
    Crc : DWORD;
END_VAR

Pos := OPENOT_WriteHeader(
    TotalLength := UINT#56,
    Flags := UINT#16#0008,
    SourceTime := SourceTime,
    RunId := RunId,
    Seq := ProducedCount,
    SourceId := SourceId,
    EventTypeId := UDINT#16#0108,
    Buffer := Buffer);

Pos := OPENOT_WriteSlotHeader(Offset := Pos, Key := UINT#16#0038, TypeTag := BYTE#16#07, PayloadLength := BYTE#8, Buffer := Buffer);
Pos := OPENOT_WriteU64LE(Offset := Pos, Value := ProducedCount, Buffer := Buffer);
Crc := OPENOT_Crc32c(Data := Buffer, Length := Pos);
Pos := OPENOT_WriteDWordLE(Offset := Pos, Value := Crc, Buffer := Buffer);
Length := Pos;
END_FUNCTION_BLOCK

(* ---- openot_value_state.st ---- *)
FUNCTION_BLOCK OPENOT_EncodeValueChangedReal
VAR_INPUT
    SourceId : UDINT;
    RunId : ULINT;
    Seq : ULINT;
    SourceTime : ULINT;
    ValueId : UDINT;
    NewValue : REAL;
    HasPrevious : BOOL;
    PreviousValue : REAL;
    HasQuality : BOOL;
    Quality : UINT;
END_VAR
VAR_OUTPUT
    Buffer : OPENOT_BYTE_BUFFER;
    Length : UINT;
END_VAR
VAR
    Pos : UINT;
    TotalLength : UINT;
    Crc : DWORD;
    ValueBits : DWORD;
END_VAR

TotalLength := UINT#60;
IF HasPrevious THEN
    TotalLength := TotalLength + UINT#8;
END_IF;
IF HasQuality THEN
    TotalLength := TotalLength + UINT#8;
END_IF;

Pos := OPENOT_WriteHeader(
    TotalLength := TotalLength,
    Flags := UINT#16#0008,
    SourceTime := SourceTime,
    RunId := RunId,
    Seq := Seq,
    SourceId := SourceId,
    EventTypeId := UDINT#16#0002,
    Buffer := Buffer);

Pos := OPENOT_WriteSlotHeader(Offset := Pos, Key := UINT#16#000D, TypeTag := BYTE#16#05, PayloadLength := BYTE#4, Buffer := Buffer);
Pos := OPENOT_WriteU32LE(Offset := Pos, Value := ValueId, Buffer := Buffer);

ValueBits := REAL_TO_DWORD(NewValue);
Pos := OPENOT_WriteSlotHeader(Offset := Pos, Key := UINT#16#0010, TypeTag := BYTE#16#09, PayloadLength := BYTE#4, Buffer := Buffer);
Pos := OPENOT_WriteDWordLE(Offset := Pos, Value := ValueBits, Buffer := Buffer);

IF HasPrevious THEN
    ValueBits := REAL_TO_DWORD(PreviousValue);
    Pos := OPENOT_WriteSlotHeader(Offset := Pos, Key := UINT#16#000F, TypeTag := BYTE#16#09, PayloadLength := BYTE#4, Buffer := Buffer);
    Pos := OPENOT_WriteDWordLE(Offset := Pos, Value := ValueBits, Buffer := Buffer);
END_IF;

IF HasQuality THEN
    Pos := OPENOT_WriteSlotHeader(Offset := Pos, Key := UINT#16#0011, TypeTag := BYTE#16#03, PayloadLength := BYTE#2, Buffer := Buffer);
    Pos := OPENOT_WriteU16LE(Offset := Pos, Value := Quality, Buffer := Buffer);
    Pos := OPENOT_WriteByte(Offset := Pos, Value := BYTE#16#00, Buffer := Buffer);
    Pos := OPENOT_WriteByte(Offset := Pos, Value := BYTE#16#00, Buffer := Buffer);
END_IF;

Crc := OPENOT_Crc32c(Data := Buffer, Length := Pos);
Pos := OPENOT_WriteDWordLE(Offset := Pos, Value := Crc, Buffer := Buffer);
Length := Pos;
END_FUNCTION_BLOCK

FUNCTION_BLOCK OPENOT_EncodeConditionLifecycle
VAR_INPUT
    SourceId : UDINT;
    RunId : ULINT;
    Seq : ULINT;
    SourceTime : ULINT;
    EventTypeId : UDINT;
    ConditionId : UDINT;
    CorrelationId : UDINT;
    HasAckBy : BOOL;
    AckBy : STRING[96];
    HasShelveSecs : BOOL;
    ShelveSecs : UDINT;
    HasReason : BOOL;
    Reason : STRING[96];
    HasComment : BOOL;
    Comment : STRING[96];
    HasPreviousPriority : BOOL;
    PreviousPriority : UINT;
    HasNewPriority : BOOL;
    NewPriority : UINT;
    HasRefreshId : BOOL;
    RefreshId : UDINT;
END_VAR
VAR_OUTPUT
    Buffer : OPENOT_BYTE_BUFFER;
    Length : UINT;
END_VAR
VAR
    Pos : UINT;
    TotalLength : UINT;
    Crc : DWORD;
    AckByLength : UINT;
    ReasonLength : UINT;
    CommentLength : UINT;
    IsActivationScoped : BOOL;
END_VAR

AckByLength := INT_TO_UINT(LEN(AckBy));
ReasonLength := INT_TO_UINT(LEN(Reason));
CommentLength := INT_TO_UINT(LEN(Comment));
IF AckByLength > UINT#96 THEN
    AckByLength := UINT#96;
END_IF;
IF ReasonLength > UINT#96 THEN
    ReasonLength := UINT#96;
END_IF;
IF CommentLength > UINT#96 THEN
    CommentLength := UINT#96;
END_IF;

IsActivationScoped := (EventTypeId = UDINT#16#0202) OR (EventTypeId = UDINT#16#0203) OR (EventTypeId = UDINT#16#0204) OR (EventTypeId = UDINT#16#0205) OR (EventTypeId = UDINT#16#020A) OR (EventTypeId = UDINT#16#020B);
TotalLength := UINT#52;
IF IsActivationScoped THEN
    TotalLength := TotalLength + UINT#8;
END_IF;
IF HasComment THEN
    TotalLength := TotalLength + OPENOT_ValueSlotEncodedLength(PayloadLength := CommentLength);
END_IF;
IF HasAckBy THEN
    TotalLength := TotalLength + OPENOT_ValueSlotEncodedLength(PayloadLength := AckByLength);
END_IF;
IF HasShelveSecs THEN
    TotalLength := TotalLength + UINT#8;
END_IF;
IF HasReason THEN
    TotalLength := TotalLength + OPENOT_ValueSlotEncodedLength(PayloadLength := ReasonLength);
END_IF;
IF HasPreviousPriority THEN
    TotalLength := TotalLength + UINT#8;
END_IF;
IF HasNewPriority THEN
    TotalLength := TotalLength + UINT#8;
END_IF;
IF HasRefreshId THEN
    TotalLength := TotalLength + UINT#8;
END_IF;

Pos := OPENOT_WriteHeader(
    TotalLength := TotalLength,
    Flags := UINT#16#0008,
    SourceTime := SourceTime,
    RunId := RunId,
    Seq := Seq,
    SourceId := SourceId,
    EventTypeId := EventTypeId,
    Buffer := Buffer);

Pos := OPENOT_WriteSlotHeader(Offset := Pos, Key := UINT#16#0005, TypeTag := BYTE#16#05, PayloadLength := BYTE#4, Buffer := Buffer);
Pos := OPENOT_WriteU32LE(Offset := Pos, Value := ConditionId, Buffer := Buffer);

IF IsActivationScoped THEN
    Pos := OPENOT_WriteSlotHeader(Offset := Pos, Key := UINT#16#0007, TypeTag := BYTE#16#05, PayloadLength := BYTE#4, Buffer := Buffer);
    Pos := OPENOT_WriteU32LE(Offset := Pos, Value := CorrelationId, Buffer := Buffer);
END_IF;

IF EventTypeId = UDINT#16#020A THEN
    IF HasComment THEN
        Pos := OPENOT_WriteSlotHeader(Offset := Pos, Key := UINT#16#0037, TypeTag := BYTE#16#0C, PayloadLength := UINT_TO_BYTE(CommentLength), Buffer := Buffer);
        Pos := OPENOT_WriteStringPayload(Offset := Pos, Value := Comment, PayloadLength := CommentLength, Buffer := Buffer);
    END_IF;

    IF HasAckBy THEN
        Pos := OPENOT_WriteSlotHeader(Offset := Pos, Key := UINT#16#001D, TypeTag := BYTE#16#0C, PayloadLength := UINT_TO_BYTE(AckByLength), Buffer := Buffer);
        Pos := OPENOT_WriteStringPayload(Offset := Pos, Value := AckBy, PayloadLength := AckByLength, Buffer := Buffer);
    END_IF;
ELSIF EventTypeId = UDINT#16#020C THEN
    IF HasPreviousPriority THEN
        Pos := OPENOT_WriteSlotHeader(Offset := Pos, Key := UINT#16#002E, TypeTag := BYTE#16#03, PayloadLength := BYTE#2, Buffer := Buffer);
        Pos := OPENOT_WriteU16LE(Offset := Pos, Value := PreviousPriority, Buffer := Buffer);
        Pos := OPENOT_WriteByte(Offset := Pos, Value := BYTE#16#00, Buffer := Buffer);
        Pos := OPENOT_WriteByte(Offset := Pos, Value := BYTE#16#00, Buffer := Buffer);
    END_IF;

    IF HasNewPriority THEN
        Pos := OPENOT_WriteSlotHeader(Offset := Pos, Key := UINT#16#002C, TypeTag := BYTE#16#03, PayloadLength := BYTE#2, Buffer := Buffer);
        Pos := OPENOT_WriteU16LE(Offset := Pos, Value := NewPriority, Buffer := Buffer);
        Pos := OPENOT_WriteByte(Offset := Pos, Value := BYTE#16#00, Buffer := Buffer);
        Pos := OPENOT_WriteByte(Offset := Pos, Value := BYTE#16#00, Buffer := Buffer);
    END_IF;

    IF HasAckBy THEN
        Pos := OPENOT_WriteSlotHeader(Offset := Pos, Key := UINT#16#001D, TypeTag := BYTE#16#0C, PayloadLength := UINT_TO_BYTE(AckByLength), Buffer := Buffer);
        Pos := OPENOT_WriteStringPayload(Offset := Pos, Value := AckBy, PayloadLength := AckByLength, Buffer := Buffer);
    END_IF;
ELSE
    IF HasAckBy THEN
        Pos := OPENOT_WriteSlotHeader(Offset := Pos, Key := UINT#16#001D, TypeTag := BYTE#16#0C, PayloadLength := UINT_TO_BYTE(AckByLength), Buffer := Buffer);
        Pos := OPENOT_WriteStringPayload(Offset := Pos, Value := AckBy, PayloadLength := AckByLength, Buffer := Buffer);
    END_IF;

    IF HasShelveSecs THEN
        Pos := OPENOT_WriteSlotHeader(Offset := Pos, Key := UINT#16#001E, TypeTag := BYTE#16#05, PayloadLength := BYTE#4, Buffer := Buffer);
        Pos := OPENOT_WriteU32LE(Offset := Pos, Value := ShelveSecs, Buffer := Buffer);
    END_IF;

    IF HasReason THEN
        Pos := OPENOT_WriteSlotHeader(Offset := Pos, Key := UINT#16#001F, TypeTag := BYTE#16#0C, PayloadLength := UINT_TO_BYTE(ReasonLength), Buffer := Buffer);
        Pos := OPENOT_WriteStringPayload(Offset := Pos, Value := Reason, PayloadLength := ReasonLength, Buffer := Buffer);
    END_IF;
END_IF;

IF HasRefreshId THEN
    Pos := OPENOT_WriteSlotHeader(Offset := Pos, Key := UINT#16#0034, TypeTag := BYTE#16#05, PayloadLength := BYTE#4, Buffer := Buffer);
    Pos := OPENOT_WriteU32LE(Offset := Pos, Value := RefreshId, Buffer := Buffer);
END_IF;

Crc := OPENOT_Crc32c(Data := Buffer, Length := Pos);
Pos := OPENOT_WriteDWordLE(Offset := Pos, Value := Crc, Buffer := Buffer);
Length := Pos;
END_FUNCTION_BLOCK

FUNCTION_BLOCK OPENOT_EncodeBatchRecipe
VAR_INPUT
    SourceId : UDINT;
    RunId : ULINT;
    Seq : ULINT;
    SourceTime : ULINT;
    EventTypeId : UDINT;
    RecipeId : UDINT;
    HasRecipeId : BOOL;
    RecipeVersion : STRING[96];
    HasBatchId : BOOL;
    BatchId : UDINT;
    HasAuthResult : BOOL;
    AuthResult : UINT;
    HasAckBy : BOOL;
    AckBy : STRING[96];
    NewState : UINT;
    MaterialId : UDINT;
    Quantity : LREAL;
    HasUnit : BOOL;
    UnitId : UINT;
END_VAR
VAR_OUTPUT
    Buffer : OPENOT_BYTE_BUFFER;
    Length : UINT;
END_VAR
VAR
    Pos : UINT;
    TotalLength : UINT;
    Crc : DWORD;
    RecipeVersionLength : UINT;
    AckByLength : UINT;
    QuantityBits : ULINT;
END_VAR

RecipeVersionLength := INT_TO_UINT(LEN(RecipeVersion));
AckByLength := INT_TO_UINT(LEN(AckBy));
IF RecipeVersionLength > UINT#96 THEN
    RecipeVersionLength := UINT#96;
END_IF;
IF AckByLength > UINT#96 THEN
    AckByLength := UINT#96;
END_IF;

IF EventTypeId = UDINT#16#0301 THEN
    TotalLength := UINT#52 + OPENOT_ValueSlotEncodedLength(PayloadLength := RecipeVersionLength);
    IF HasBatchId THEN
        TotalLength := TotalLength + UINT#8;
    END_IF;
ELSIF EventTypeId = UDINT#16#0302 THEN
    TotalLength := UINT#52 + OPENOT_ValueSlotEncodedLength(PayloadLength := RecipeVersionLength);
    IF HasAuthResult THEN
        TotalLength := TotalLength + UINT#8;
    END_IF;
    IF HasAckBy THEN
        TotalLength := TotalLength + OPENOT_ValueSlotEncodedLength(PayloadLength := AckByLength);
    END_IF;
ELSIF EventTypeId = UDINT#16#0303 THEN
    TotalLength := UINT#60;
    IF HasRecipeId THEN
        TotalLength := TotalLength + UINT#8;
    END_IF;
ELSIF EventTypeId = UDINT#16#0304 THEN
    TotalLength := UINT#72;
    IF HasUnit THEN
        TotalLength := TotalLength + UINT#8;
    END_IF;
ELSE
    TotalLength := UINT#0;
END_IF;

IF TotalLength > UINT#0 THEN
    Pos := OPENOT_WriteHeader(
        TotalLength := TotalLength,
        Flags := UINT#16#0008,
        SourceTime := SourceTime,
        RunId := RunId,
        Seq := Seq,
        SourceId := SourceId,
        EventTypeId := EventTypeId,
        Buffer := Buffer);

    IF EventTypeId = UDINT#16#0301 THEN
        Pos := OPENOT_WriteSlotHeader(Offset := Pos, Key := UINT#16#0023, TypeTag := BYTE#16#05, PayloadLength := BYTE#4, Buffer := Buffer);
        Pos := OPENOT_WriteU32LE(Offset := Pos, Value := RecipeId, Buffer := Buffer);
        Pos := OPENOT_WriteSlotHeader(Offset := Pos, Key := UINT#16#0024, TypeTag := BYTE#16#0C, PayloadLength := UINT_TO_BYTE(RecipeVersionLength), Buffer := Buffer);
        Pos := OPENOT_WriteStringPayload(Offset := Pos, Value := RecipeVersion, PayloadLength := RecipeVersionLength, Buffer := Buffer);
        IF HasBatchId THEN
            Pos := OPENOT_WriteSlotHeader(Offset := Pos, Key := UINT#16#0025, TypeTag := BYTE#16#05, PayloadLength := BYTE#4, Buffer := Buffer);
            Pos := OPENOT_WriteU32LE(Offset := Pos, Value := BatchId, Buffer := Buffer);
        END_IF;
    ELSIF EventTypeId = UDINT#16#0302 THEN
        Pos := OPENOT_WriteSlotHeader(Offset := Pos, Key := UINT#16#0023, TypeTag := BYTE#16#05, PayloadLength := BYTE#4, Buffer := Buffer);
        Pos := OPENOT_WriteU32LE(Offset := Pos, Value := RecipeId, Buffer := Buffer);
        Pos := OPENOT_WriteSlotHeader(Offset := Pos, Key := UINT#16#0024, TypeTag := BYTE#16#0C, PayloadLength := UINT_TO_BYTE(RecipeVersionLength), Buffer := Buffer);
        Pos := OPENOT_WriteStringPayload(Offset := Pos, Value := RecipeVersion, PayloadLength := RecipeVersionLength, Buffer := Buffer);
        IF HasAuthResult THEN
            Pos := OPENOT_WriteSlotHeader(Offset := Pos, Key := UINT#16#0020, TypeTag := BYTE#16#03, PayloadLength := BYTE#2, Buffer := Buffer);
            Pos := OPENOT_WriteU16LE(Offset := Pos, Value := AuthResult, Buffer := Buffer);
            Pos := OPENOT_WriteByte(Offset := Pos, Value := BYTE#16#00, Buffer := Buffer);
            Pos := OPENOT_WriteByte(Offset := Pos, Value := BYTE#16#00, Buffer := Buffer);
        END_IF;
        IF HasAckBy THEN
            Pos := OPENOT_WriteSlotHeader(Offset := Pos, Key := UINT#16#001D, TypeTag := BYTE#16#0C, PayloadLength := UINT_TO_BYTE(AckByLength), Buffer := Buffer);
            Pos := OPENOT_WriteStringPayload(Offset := Pos, Value := AckBy, PayloadLength := AckByLength, Buffer := Buffer);
        END_IF;
    ELSIF EventTypeId = UDINT#16#0303 THEN
        Pos := OPENOT_WriteSlotHeader(Offset := Pos, Key := UINT#16#0025, TypeTag := BYTE#16#05, PayloadLength := BYTE#4, Buffer := Buffer);
        Pos := OPENOT_WriteU32LE(Offset := Pos, Value := BatchId, Buffer := Buffer);
        Pos := OPENOT_WriteSlotHeader(Offset := Pos, Key := UINT#16#0004, TypeTag := BYTE#16#03, PayloadLength := BYTE#2, Buffer := Buffer);
        Pos := OPENOT_WriteU16LE(Offset := Pos, Value := NewState, Buffer := Buffer);
        Pos := OPENOT_WriteByte(Offset := Pos, Value := BYTE#16#00, Buffer := Buffer);
        Pos := OPENOT_WriteByte(Offset := Pos, Value := BYTE#16#00, Buffer := Buffer);
        IF HasRecipeId THEN
            Pos := OPENOT_WriteSlotHeader(Offset := Pos, Key := UINT#16#0023, TypeTag := BYTE#16#05, PayloadLength := BYTE#4, Buffer := Buffer);
            Pos := OPENOT_WriteU32LE(Offset := Pos, Value := RecipeId, Buffer := Buffer);
        END_IF;
    ELSIF EventTypeId = UDINT#16#0304 THEN
        Pos := OPENOT_WriteSlotHeader(Offset := Pos, Key := UINT#16#0025, TypeTag := BYTE#16#05, PayloadLength := BYTE#4, Buffer := Buffer);
        Pos := OPENOT_WriteU32LE(Offset := Pos, Value := BatchId, Buffer := Buffer);
        Pos := OPENOT_WriteSlotHeader(Offset := Pos, Key := UINT#16#0026, TypeTag := BYTE#16#05, PayloadLength := BYTE#4, Buffer := Buffer);
        Pos := OPENOT_WriteU32LE(Offset := Pos, Value := MaterialId, Buffer := Buffer);
        QuantityBits := LWORD_TO_ULINT(LREAL_TO_LWORD(Quantity));
        Pos := OPENOT_WriteSlotHeader(Offset := Pos, Key := UINT#16#0027, TypeTag := BYTE#16#0A, PayloadLength := BYTE#8, Buffer := Buffer);
        Pos := OPENOT_WriteU64LE(Offset := Pos, Value := QuantityBits, Buffer := Buffer);
        IF HasUnit THEN
            Pos := OPENOT_WriteSlotHeader(Offset := Pos, Key := UINT#16#0013, TypeTag := BYTE#16#03, PayloadLength := BYTE#2, Buffer := Buffer);
            Pos := OPENOT_WriteU16LE(Offset := Pos, Value := UnitId, Buffer := Buffer);
            Pos := OPENOT_WriteByte(Offset := Pos, Value := BYTE#16#00, Buffer := Buffer);
            Pos := OPENOT_WriteByte(Offset := Pos, Value := BYTE#16#00, Buffer := Buffer);
        END_IF;
    END_IF;

    Crc := OPENOT_Crc32c(Data := Buffer, Length := Pos);
    Pos := OPENOT_WriteDWordLE(Offset := Pos, Value := Crc, Buffer := Buffer);
    Length := Pos;
ELSE
    Length := UINT#0;
END_IF;
END_FUNCTION_BLOCK

FUNCTION_BLOCK OPENOT_EncodeConformantConditionAcknowledged
VAR_OUTPUT
    Buffer : OPENOT_BYTE_BUFFER;
    Length : UINT;
END_VAR
VAR
    Encoder : OPENOT_EncodeConditionLifecycle;
END_VAR

Encoder(
    SourceId := UDINT#66,
    RunId := ULINT#1,
    Seq := ULINT#17,
    SourceTime := ULINT#1000000160,
    EventTypeId := UDINT#16#0202,
    ConditionId := UDINT#9001,
    CorrelationId := UDINT#77,
    HasAckBy := TRUE,
    AckBy := 'operator-a',
    HasShelveSecs := FALSE,
    ShelveSecs := UDINT#0,
    HasReason := FALSE,
    Reason := '',
    HasComment := FALSE,
    Comment := '',
    HasPreviousPriority := FALSE,
    PreviousPriority := UINT#0,
    HasNewPriority := FALSE,
    NewPriority := UINT#0,
    HasRefreshId := FALSE,
    RefreshId := UDINT#0);
Buffer := Encoder.Buffer;
Length := Encoder.Length;
END_FUNCTION_BLOCK

FUNCTION_BLOCK OPENOT_EncodeConformantConditionShelved
VAR_OUTPUT
    Buffer : OPENOT_BYTE_BUFFER;
    Length : UINT;
END_VAR
VAR
    Encoder : OPENOT_EncodeConditionLifecycle;
END_VAR

Encoder(
    SourceId := UDINT#66,
    RunId := ULINT#1,
    Seq := ULINT#18,
    SourceTime := ULINT#1000000170,
    EventTypeId := UDINT#16#0204,
    ConditionId := UDINT#9001,
    CorrelationId := UDINT#77,
    HasAckBy := TRUE,
    AckBy := 'operator-a',
    HasShelveSecs := TRUE,
    ShelveSecs := UDINT#300,
    HasReason := FALSE,
    Reason := '',
    HasComment := FALSE,
    Comment := '',
    HasPreviousPriority := FALSE,
    PreviousPriority := UINT#0,
    HasNewPriority := FALSE,
    NewPriority := UINT#0,
    HasRefreshId := FALSE,
    RefreshId := UDINT#0);
Buffer := Encoder.Buffer;
Length := Encoder.Length;
END_FUNCTION_BLOCK

FUNCTION_BLOCK OPENOT_EncodeConformantConditionSuppressed
VAR_OUTPUT
    Buffer : OPENOT_BYTE_BUFFER;
    Length : UINT;
END_VAR
VAR
    Encoder : OPENOT_EncodeConditionLifecycle;
END_VAR

Encoder(
    SourceId := UDINT#66,
    RunId := ULINT#1,
    Seq := ULINT#19,
    SourceTime := ULINT#1000000180,
    EventTypeId := UDINT#16#0206,
    ConditionId := UDINT#9001,
    CorrelationId := UDINT#0,
    HasAckBy := FALSE,
    AckBy := '',
    HasShelveSecs := FALSE,
    ShelveSecs := UDINT#0,
    HasReason := TRUE,
    Reason := 'maintenance',
    HasComment := FALSE,
    Comment := '',
    HasPreviousPriority := FALSE,
    PreviousPriority := UINT#0,
    HasNewPriority := FALSE,
    NewPriority := UINT#0,
    HasRefreshId := FALSE,
    RefreshId := UDINT#0);
Buffer := Encoder.Buffer;
Length := Encoder.Length;
END_FUNCTION_BLOCK

FUNCTION_BLOCK OPENOT_EncodeConformantConditionOutOfService
VAR_OUTPUT
    Buffer : OPENOT_BYTE_BUFFER;
    Length : UINT;
END_VAR
VAR
    Encoder : OPENOT_EncodeConditionLifecycle;
END_VAR

Encoder(
    SourceId := UDINT#66,
    RunId := ULINT#1,
    Seq := ULINT#20,
    SourceTime := ULINT#1000000190,
    EventTypeId := UDINT#16#0208,
    ConditionId := UDINT#9001,
    CorrelationId := UDINT#0,
    HasAckBy := TRUE,
    AckBy := 'operator-a',
    HasShelveSecs := FALSE,
    ShelveSecs := UDINT#0,
    HasReason := FALSE,
    Reason := '',
    HasComment := FALSE,
    Comment := '',
    HasPreviousPriority := FALSE,
    PreviousPriority := UINT#0,
    HasNewPriority := FALSE,
    NewPriority := UINT#0,
    HasRefreshId := FALSE,
    RefreshId := UDINT#0);
Buffer := Encoder.Buffer;
Length := Encoder.Length;
END_FUNCTION_BLOCK

FUNCTION_BLOCK OPENOT_EncodeConformantConditionConfirmed
VAR_OUTPUT
    Buffer : OPENOT_BYTE_BUFFER;
    Length : UINT;
END_VAR
VAR
    Encoder : OPENOT_EncodeConditionLifecycle;
END_VAR

Encoder(
    SourceId := UDINT#66,
    RunId := ULINT#1,
    Seq := ULINT#21,
    SourceTime := ULINT#1000000200,
    EventTypeId := UDINT#16#0203,
    ConditionId := UDINT#9001,
    CorrelationId := UDINT#77,
    HasAckBy := TRUE,
    AckBy := 'operator-a',
    HasShelveSecs := FALSE,
    ShelveSecs := UDINT#0,
    HasReason := FALSE,
    Reason := '',
    HasComment := FALSE,
    Comment := '',
    HasPreviousPriority := FALSE,
    PreviousPriority := UINT#0,
    HasNewPriority := FALSE,
    NewPriority := UINT#0,
    HasRefreshId := FALSE,
    RefreshId := UDINT#0);
Buffer := Encoder.Buffer;
Length := Encoder.Length;
END_FUNCTION_BLOCK

FUNCTION_BLOCK OPENOT_EncodeConformantConditionUnshelved
VAR_OUTPUT
    Buffer : OPENOT_BYTE_BUFFER;
    Length : UINT;
END_VAR
VAR
    Encoder : OPENOT_EncodeConditionLifecycle;
END_VAR

Encoder(
    SourceId := UDINT#66,
    RunId := ULINT#1,
    Seq := ULINT#22,
    SourceTime := ULINT#1000000210,
    EventTypeId := UDINT#16#0205,
    ConditionId := UDINT#9001,
    CorrelationId := UDINT#77,
    HasAckBy := FALSE,
    AckBy := '',
    HasShelveSecs := FALSE,
    ShelveSecs := UDINT#0,
    HasReason := FALSE,
    Reason := '',
    HasComment := FALSE,
    Comment := '',
    HasPreviousPriority := FALSE,
    PreviousPriority := UINT#0,
    HasNewPriority := FALSE,
    NewPriority := UINT#0,
    HasRefreshId := FALSE,
    RefreshId := UDINT#0);
Buffer := Encoder.Buffer;
Length := Encoder.Length;
END_FUNCTION_BLOCK

FUNCTION_BLOCK OPENOT_EncodeConformantConditionUnsuppressed
VAR_OUTPUT
    Buffer : OPENOT_BYTE_BUFFER;
    Length : UINT;
END_VAR
VAR
    Encoder : OPENOT_EncodeConditionLifecycle;
END_VAR

Encoder(
    SourceId := UDINT#66,
    RunId := ULINT#1,
    Seq := ULINT#23,
    SourceTime := ULINT#1000000220,
    EventTypeId := UDINT#16#0207,
    ConditionId := UDINT#9001,
    CorrelationId := UDINT#0,
    HasAckBy := FALSE,
    AckBy := '',
    HasShelveSecs := FALSE,
    ShelveSecs := UDINT#0,
    HasReason := FALSE,
    Reason := '',
    HasComment := FALSE,
    Comment := '',
    HasPreviousPriority := FALSE,
    PreviousPriority := UINT#0,
    HasNewPriority := FALSE,
    NewPriority := UINT#0,
    HasRefreshId := FALSE,
    RefreshId := UDINT#0);
Buffer := Encoder.Buffer;
Length := Encoder.Length;
END_FUNCTION_BLOCK

FUNCTION_BLOCK OPENOT_EncodeConformantConditionInService
VAR_OUTPUT
    Buffer : OPENOT_BYTE_BUFFER;
    Length : UINT;
END_VAR
VAR
    Encoder : OPENOT_EncodeConditionLifecycle;
END_VAR

Encoder(
    SourceId := UDINT#66,
    RunId := ULINT#1,
    Seq := ULINT#24,
    SourceTime := ULINT#1000000230,
    EventTypeId := UDINT#16#0209,
    ConditionId := UDINT#9001,
    CorrelationId := UDINT#0,
    HasAckBy := FALSE,
    AckBy := '',
    HasShelveSecs := FALSE,
    ShelveSecs := UDINT#0,
    HasReason := FALSE,
    Reason := '',
    HasComment := FALSE,
    Comment := '',
    HasPreviousPriority := FALSE,
    PreviousPriority := UINT#0,
    HasNewPriority := FALSE,
    NewPriority := UINT#0,
    HasRefreshId := FALSE,
    RefreshId := UDINT#0);
Buffer := Encoder.Buffer;
Length := Encoder.Length;
END_FUNCTION_BLOCK

FUNCTION_BLOCK OPENOT_EncodeConformantConditionReset
VAR_OUTPUT
    Buffer : OPENOT_BYTE_BUFFER;
    Length : UINT;
END_VAR
VAR
    Encoder : OPENOT_EncodeConditionLifecycle;
END_VAR

Encoder(
    SourceId := UDINT#66,
    RunId := ULINT#1,
    Seq := ULINT#25,
    SourceTime := ULINT#1000000240,
    EventTypeId := UDINT#16#020B,
    ConditionId := UDINT#9001,
    CorrelationId := UDINT#77,
    HasAckBy := TRUE,
    AckBy := 'operator-a',
    HasShelveSecs := FALSE,
    ShelveSecs := UDINT#0,
    HasReason := FALSE,
    Reason := '',
    HasComment := FALSE,
    Comment := '',
    HasPreviousPriority := FALSE,
    PreviousPriority := UINT#0,
    HasNewPriority := FALSE,
    NewPriority := UINT#0,
    HasRefreshId := FALSE,
    RefreshId := UDINT#0);
Buffer := Encoder.Buffer;
Length := Encoder.Length;
END_FUNCTION_BLOCK

FUNCTION_BLOCK OPENOT_EncodeConformantConditionCommented
VAR_OUTPUT
    Buffer : OPENOT_BYTE_BUFFER;
    Length : UINT;
END_VAR
VAR
    Encoder : OPENOT_EncodeConditionLifecycle;
END_VAR

Encoder(
    SourceId := UDINT#66,
    RunId := ULINT#1,
    Seq := ULINT#26,
    SourceTime := ULINT#1000000250,
    EventTypeId := UDINT#16#020A,
    ConditionId := UDINT#9001,
    CorrelationId := UDINT#77,
    HasAckBy := TRUE,
    AckBy := 'operator-a',
    HasShelveSecs := FALSE,
    ShelveSecs := UDINT#0,
    HasReason := FALSE,
    Reason := '',
    HasComment := TRUE,
    Comment := 'operator comment',
    HasPreviousPriority := FALSE,
    PreviousPriority := UINT#0,
    HasNewPriority := FALSE,
    NewPriority := UINT#0,
    HasRefreshId := FALSE,
    RefreshId := UDINT#0);
Buffer := Encoder.Buffer;
Length := Encoder.Length;
END_FUNCTION_BLOCK

FUNCTION_BLOCK OPENOT_EncodeConformantConditionPriorityChanged
VAR_OUTPUT
    Buffer : OPENOT_BYTE_BUFFER;
    Length : UINT;
END_VAR
VAR
    Encoder : OPENOT_EncodeConditionLifecycle;
END_VAR

Encoder(
    SourceId := UDINT#66,
    RunId := ULINT#1,
    Seq := ULINT#27,
    SourceTime := ULINT#1000000260,
    EventTypeId := UDINT#16#020C,
    ConditionId := UDINT#9001,
    CorrelationId := UDINT#0,
    HasAckBy := TRUE,
    AckBy := 'operator-a',
    HasShelveSecs := FALSE,
    ShelveSecs := UDINT#0,
    HasReason := FALSE,
    Reason := '',
    HasComment := FALSE,
    Comment := '',
    HasPreviousPriority := TRUE,
    PreviousPriority := UINT#600,
    HasNewPriority := TRUE,
    NewPriority := UINT#900,
    HasRefreshId := FALSE,
    RefreshId := UDINT#0);
Buffer := Encoder.Buffer;
Length := Encoder.Length;
END_FUNCTION_BLOCK

FUNCTION_BLOCK OPENOT_EncodeConformantRecipeLoaded
VAR_OUTPUT
    Buffer : OPENOT_BYTE_BUFFER;
    Length : UINT;
END_VAR
VAR
    Encoder : OPENOT_EncodeBatchRecipe;
END_VAR

Encoder(
    SourceId := UDINT#66,
    RunId := ULINT#1,
    Seq := ULINT#28,
    SourceTime := ULINT#1000000270,
    EventTypeId := UDINT#16#0301,
    RecipeId := UDINT#3001,
    HasRecipeId := TRUE,
    RecipeVersion := 'v1.2.3',
    HasBatchId := TRUE,
    BatchId := UDINT#4001,
    HasAuthResult := FALSE,
    AuthResult := UINT#0,
    HasAckBy := FALSE,
    AckBy := '',
    NewState := UINT#0,
    MaterialId := UDINT#0,
    Quantity := LREAL#0.0,
    HasUnit := FALSE,
    UnitId := UINT#0);
Buffer := Encoder.Buffer;
Length := Encoder.Length;
END_FUNCTION_BLOCK

FUNCTION_BLOCK OPENOT_EncodeConformantRecipeApproved
VAR_OUTPUT
    Buffer : OPENOT_BYTE_BUFFER;
    Length : UINT;
END_VAR
VAR
    Encoder : OPENOT_EncodeBatchRecipe;
END_VAR

Encoder(
    SourceId := UDINT#66,
    RunId := ULINT#1,
    Seq := ULINT#29,
    SourceTime := ULINT#1000000280,
    EventTypeId := UDINT#16#0302,
    RecipeId := UDINT#3001,
    HasRecipeId := TRUE,
    RecipeVersion := 'v1.2.3',
    HasBatchId := FALSE,
    BatchId := UDINT#0,
    HasAuthResult := TRUE,
    AuthResult := UINT#1,
    HasAckBy := TRUE,
    AckBy := 'approver-a',
    NewState := UINT#0,
    MaterialId := UDINT#0,
    Quantity := LREAL#0.0,
    HasUnit := FALSE,
    UnitId := UINT#0);
Buffer := Encoder.Buffer;
Length := Encoder.Length;
END_FUNCTION_BLOCK

FUNCTION_BLOCK OPENOT_EncodeConformantBatchEvent
VAR_OUTPUT
    Buffer : OPENOT_BYTE_BUFFER;
    Length : UINT;
END_VAR
VAR
    Encoder : OPENOT_EncodeBatchRecipe;
END_VAR

Encoder(
    SourceId := UDINT#66,
    RunId := ULINT#1,
    Seq := ULINT#30,
    SourceTime := ULINT#1000000290,
    EventTypeId := UDINT#16#0303,
    RecipeId := UDINT#3001,
    HasRecipeId := TRUE,
    RecipeVersion := '',
    HasBatchId := TRUE,
    BatchId := UDINT#4001,
    HasAuthResult := FALSE,
    AuthResult := UINT#0,
    HasAckBy := FALSE,
    AckBy := '',
    NewState := UINT#2,
    MaterialId := UDINT#0,
    Quantity := LREAL#0.0,
    HasUnit := FALSE,
    UnitId := UINT#0);
Buffer := Encoder.Buffer;
Length := Encoder.Length;
END_FUNCTION_BLOCK

FUNCTION_BLOCK OPENOT_EncodeConformantMaterialAddition
VAR_OUTPUT
    Buffer : OPENOT_BYTE_BUFFER;
    Length : UINT;
END_VAR
VAR
    Encoder : OPENOT_EncodeBatchRecipe;
END_VAR

Encoder(
    SourceId := UDINT#66,
    RunId := ULINT#1,
    Seq := ULINT#31,
    SourceTime := ULINT#1000000300,
    EventTypeId := UDINT#16#0304,
    RecipeId := UDINT#0,
    HasRecipeId := FALSE,
    RecipeVersion := '',
    HasBatchId := TRUE,
    BatchId := UDINT#4001,
    HasAuthResult := FALSE,
    AuthResult := UINT#0,
    HasAckBy := FALSE,
    AckBy := '',
    NewState := UINT#0,
    MaterialId := UDINT#5001,
    Quantity := LREAL#12.25,
    HasUnit := TRUE,
    UnitId := UINT#8);
Buffer := Encoder.Buffer;
Length := Encoder.Length;
END_FUNCTION_BLOCK

FUNCTION_BLOCK OPENOT_EncodeValueChangedInt
VAR_INPUT
    SourceId : UDINT;
    RunId : ULINT;
    Seq : ULINT;
    SourceTime : ULINT;
    ValueId : UDINT;
    NewValue : DINT;
    HasPrevious : BOOL;
    PreviousValue : DINT;
    HasQuality : BOOL;
    Quality : UINT;
END_VAR
VAR_OUTPUT
    Buffer : OPENOT_BYTE_BUFFER;
    Length : UINT;
END_VAR
VAR
    Pos : UINT;
    TotalLength : UINT;
    Crc : DWORD;
    ValueBits : DWORD;
END_VAR

TotalLength := UINT#60;
IF HasPrevious THEN
    TotalLength := TotalLength + UINT#8;
END_IF;
IF HasQuality THEN
    TotalLength := TotalLength + UINT#8;
END_IF;

Pos := OPENOT_WriteHeader(
    TotalLength := TotalLength,
    Flags := UINT#16#0008,
    SourceTime := SourceTime,
    RunId := RunId,
    Seq := Seq,
    SourceId := SourceId,
    EventTypeId := UDINT#16#0002,
    Buffer := Buffer);

Pos := OPENOT_WriteSlotHeader(Offset := Pos, Key := UINT#16#000D, TypeTag := BYTE#16#05, PayloadLength := BYTE#4, Buffer := Buffer);
Pos := OPENOT_WriteU32LE(Offset := Pos, Value := ValueId, Buffer := Buffer);

ValueBits := DINT_TO_DWORD(NewValue);
Pos := OPENOT_WriteSlotHeader(Offset := Pos, Key := UINT#16#0010, TypeTag := BYTE#16#06, PayloadLength := BYTE#4, Buffer := Buffer);
Pos := OPENOT_WriteDWordLE(Offset := Pos, Value := ValueBits, Buffer := Buffer);

IF HasPrevious THEN
    ValueBits := DINT_TO_DWORD(PreviousValue);
    Pos := OPENOT_WriteSlotHeader(Offset := Pos, Key := UINT#16#000F, TypeTag := BYTE#16#06, PayloadLength := BYTE#4, Buffer := Buffer);
    Pos := OPENOT_WriteDWordLE(Offset := Pos, Value := ValueBits, Buffer := Buffer);
END_IF;

IF HasQuality THEN
    Pos := OPENOT_WriteSlotHeader(Offset := Pos, Key := UINT#16#0011, TypeTag := BYTE#16#03, PayloadLength := BYTE#2, Buffer := Buffer);
    Pos := OPENOT_WriteU16LE(Offset := Pos, Value := Quality, Buffer := Buffer);
    Pos := OPENOT_WriteByte(Offset := Pos, Value := BYTE#16#00, Buffer := Buffer);
    Pos := OPENOT_WriteByte(Offset := Pos, Value := BYTE#16#00, Buffer := Buffer);
END_IF;

Crc := OPENOT_Crc32c(Data := Buffer, Length := Pos);
Pos := OPENOT_WriteDWordLE(Offset := Pos, Value := Crc, Buffer := Buffer);
Length := Pos;
END_FUNCTION_BLOCK

FUNCTION OPENOT_ValueSlotEncodedLength : UINT
VAR_INPUT
    PayloadLength : UINT;
END_VAR
VAR
    Padding : UINT;
END_VAR

Padding := UINT#0;
IF (PayloadLength MOD UINT#4) <> UINT#0 THEN
    Padding := UINT#4 - (PayloadLength MOD UINT#4);
END_IF;

OPENOT_ValueSlotEncodedLength := UINT#4 + PayloadLength + Padding;
END_FUNCTION

FUNCTION OPENOT_WriteValueBitsLE : UINT
VAR_INPUT
    Offset : UINT;
    Value : ULINT;
    PayloadLength : UINT;
END_VAR
VAR_IN_OUT
    Buffer : OPENOT_BYTE_BUFFER;
END_VAR
VAR
    Remaining : ULINT;
    Index : UINT;
    Pos : UINT;
END_VAR

Remaining := Value;
Pos := Offset;
FOR Index := UINT#0 TO PayloadLength - UINT#1 DO
    Pos := OPENOT_WriteByte(Offset := Pos, Value := ULINT_TO_BYTE(Remaining MOD ULINT#256), Buffer := Buffer);
    Remaining := Remaining / ULINT#256;
END_FOR;
WHILE (Pos MOD UINT#4) <> UINT#0 DO
    Pos := OPENOT_WriteByte(Offset := Pos, Value := BYTE#16#00, Buffer := Buffer);
END_WHILE;
OPENOT_WriteValueBitsLE := Pos;
END_FUNCTION

FUNCTION_BLOCK OPENOT_EncodeValueChangedBits
VAR_INPUT
    SourceId : UDINT;
    RunId : ULINT;
    Seq : ULINT;
    SourceTime : ULINT;
    ValueId : UDINT;
    TypeTag : BYTE;
    PayloadLength : UINT;
    NewBits : ULINT;
    HasPrevious : BOOL;
    PreviousBits : ULINT;
    HasQuality : BOOL;
    Quality : UINT;
END_VAR
VAR_OUTPUT
    Buffer : OPENOT_BYTE_BUFFER;
    Length : UINT;
END_VAR
VAR
    Pos : UINT;
    TotalLength : UINT;
    Crc : DWORD;
END_VAR

TotalLength := UINT#40 + UINT#8 + OPENOT_ValueSlotEncodedLength(PayloadLength := PayloadLength) + UINT#4;
IF HasPrevious THEN
    TotalLength := TotalLength + OPENOT_ValueSlotEncodedLength(PayloadLength := PayloadLength);
END_IF;
IF HasQuality THEN
    TotalLength := TotalLength + UINT#8;
END_IF;

Pos := OPENOT_WriteHeader(
    TotalLength := TotalLength,
    Flags := UINT#16#0008,
    SourceTime := SourceTime,
    RunId := RunId,
    Seq := Seq,
    SourceId := SourceId,
    EventTypeId := UDINT#16#0002,
    Buffer := Buffer);

Pos := OPENOT_WriteSlotHeader(Offset := Pos, Key := UINT#16#000D, TypeTag := BYTE#16#05, PayloadLength := BYTE#4, Buffer := Buffer);
Pos := OPENOT_WriteU32LE(Offset := Pos, Value := ValueId, Buffer := Buffer);

Pos := OPENOT_WriteSlotHeader(Offset := Pos, Key := UINT#16#0010, TypeTag := TypeTag, PayloadLength := UINT_TO_BYTE(PayloadLength), Buffer := Buffer);
Pos := OPENOT_WriteValueBitsLE(Offset := Pos, Value := NewBits, PayloadLength := PayloadLength, Buffer := Buffer);

IF HasPrevious THEN
    Pos := OPENOT_WriteSlotHeader(Offset := Pos, Key := UINT#16#000F, TypeTag := TypeTag, PayloadLength := UINT_TO_BYTE(PayloadLength), Buffer := Buffer);
    Pos := OPENOT_WriteValueBitsLE(Offset := Pos, Value := PreviousBits, PayloadLength := PayloadLength, Buffer := Buffer);
END_IF;

IF HasQuality THEN
    Pos := OPENOT_WriteSlotHeader(Offset := Pos, Key := UINT#16#0011, TypeTag := BYTE#16#03, PayloadLength := BYTE#2, Buffer := Buffer);
    Pos := OPENOT_WriteU16LE(Offset := Pos, Value := Quality, Buffer := Buffer);
    Pos := OPENOT_WriteByte(Offset := Pos, Value := BYTE#16#00, Buffer := Buffer);
    Pos := OPENOT_WriteByte(Offset := Pos, Value := BYTE#16#00, Buffer := Buffer);
END_IF;

Crc := OPENOT_Crc32c(Data := Buffer, Length := Pos);
Pos := OPENOT_WriteDWordLE(Offset := Pos, Value := Crc, Buffer := Buffer);
Length := Pos;
END_FUNCTION_BLOCK

FUNCTION OPENOT_WriteStringPayload : UINT
VAR_INPUT
    Offset : UINT;
    Value : STRING[96];
    PayloadLength : UINT;
END_VAR
VAR_IN_OUT
    Buffer : OPENOT_BYTE_BUFFER;
END_VAR
VAR
    Index : UINT;
    Pos : UINT;
    Slice : STRING[1];
END_VAR

Pos := Offset;
IF PayloadLength > UINT#0 THEN
    FOR Index := UINT#0 TO PayloadLength - UINT#1 DO
        Slice := MID(IN := Value, L := INT#1, P := UINT_TO_INT(Index + UINT#1));
        Pos := OPENOT_WriteByte(Offset := Pos, Value := CHAR_TO_BYTE(STRING_TO_CHAR(Slice)), Buffer := Buffer);
    END_FOR;
END_IF;
WHILE (Pos MOD UINT#4) <> UINT#0 DO
    Pos := OPENOT_WriteByte(Offset := Pos, Value := BYTE#16#00, Buffer := Buffer);
END_WHILE;
OPENOT_WriteStringPayload := Pos;
END_FUNCTION

FUNCTION_BLOCK OPENOT_EncodeValueChangedString
VAR_INPUT
    SourceId : UDINT;
    RunId : ULINT;
    Seq : ULINT;
    SourceTime : ULINT;
    ValueId : UDINT;
    NewValue : STRING[96];
    HasPrevious : BOOL;
    PreviousValue : STRING[96];
    HasQuality : BOOL;
    Quality : UINT;
END_VAR
VAR_OUTPUT
    Buffer : OPENOT_BYTE_BUFFER;
    Length : UINT;
END_VAR
VAR
    Pos : UINT;
    TotalLength : UINT;
    NewLength : UINT;
    PreviousLength : UINT;
    Crc : DWORD;
END_VAR

NewLength := INT_TO_UINT(LEN(NewValue));
PreviousLength := INT_TO_UINT(LEN(PreviousValue));
IF NewLength > UINT#96 THEN
    NewLength := UINT#96;
END_IF;
IF PreviousLength > UINT#96 THEN
    PreviousLength := UINT#96;
END_IF;

TotalLength := UINT#40 + UINT#8 + OPENOT_ValueSlotEncodedLength(PayloadLength := NewLength) + UINT#4;
IF HasPrevious THEN
    TotalLength := TotalLength + OPENOT_ValueSlotEncodedLength(PayloadLength := PreviousLength);
END_IF;
IF HasQuality THEN
    TotalLength := TotalLength + UINT#8;
END_IF;

Pos := OPENOT_WriteHeader(
    TotalLength := TotalLength,
    Flags := UINT#16#0008,
    SourceTime := SourceTime,
    RunId := RunId,
    Seq := Seq,
    SourceId := SourceId,
    EventTypeId := UDINT#16#0002,
    Buffer := Buffer);

Pos := OPENOT_WriteSlotHeader(Offset := Pos, Key := UINT#16#000D, TypeTag := BYTE#16#05, PayloadLength := BYTE#4, Buffer := Buffer);
Pos := OPENOT_WriteU32LE(Offset := Pos, Value := ValueId, Buffer := Buffer);

Pos := OPENOT_WriteSlotHeader(Offset := Pos, Key := UINT#16#0010, TypeTag := BYTE#16#0C, PayloadLength := UINT_TO_BYTE(NewLength), Buffer := Buffer);
Pos := OPENOT_WriteStringPayload(Offset := Pos, Value := NewValue, PayloadLength := NewLength, Buffer := Buffer);

IF HasPrevious THEN
    Pos := OPENOT_WriteSlotHeader(Offset := Pos, Key := UINT#16#000F, TypeTag := BYTE#16#0C, PayloadLength := UINT_TO_BYTE(PreviousLength), Buffer := Buffer);
    Pos := OPENOT_WriteStringPayload(Offset := Pos, Value := PreviousValue, PayloadLength := PreviousLength, Buffer := Buffer);
END_IF;

IF HasQuality THEN
    Pos := OPENOT_WriteSlotHeader(Offset := Pos, Key := UINT#16#0011, TypeTag := BYTE#16#03, PayloadLength := BYTE#2, Buffer := Buffer);
    Pos := OPENOT_WriteU16LE(Offset := Pos, Value := Quality, Buffer := Buffer);
    Pos := OPENOT_WriteByte(Offset := Pos, Value := BYTE#16#00, Buffer := Buffer);
    Pos := OPENOT_WriteByte(Offset := Pos, Value := BYTE#16#00, Buffer := Buffer);
END_IF;

Crc := OPENOT_Crc32c(Data := Buffer, Length := Pos);
Pos := OPENOT_WriteDWordLE(Offset := Pos, Value := Crc, Buffer := Buffer);
Length := Pos;
END_FUNCTION_BLOCK

FUNCTION_BLOCK OPENOT_EncodeStateTransition
VAR_INPUT
    SourceId : UDINT;
    RunId : ULINT;
    Seq : ULINT;
    SourceTime : ULINT;
    StateMachineId : UDINT;
    Category : UINT;
    PreviousState : UINT;
    NewState : UINT;
END_VAR
VAR_OUTPUT
    Buffer : OPENOT_BYTE_BUFFER;
    Length : UINT;
END_VAR
VAR
    Pos : UINT;
    Crc : DWORD;
END_VAR

Pos := OPENOT_WriteHeader(
    TotalLength := UINT#76,
    Flags := UINT#16#0008,
    SourceTime := SourceTime,
    RunId := RunId,
    Seq := Seq,
    SourceId := SourceId,
    EventTypeId := UDINT#16#0001,
    Buffer := Buffer);

Pos := OPENOT_WriteSlotHeader(Offset := Pos, Key := UINT#16#0001, TypeTag := BYTE#16#05, PayloadLength := BYTE#4, Buffer := Buffer);
Pos := OPENOT_WriteU32LE(Offset := Pos, Value := StateMachineId, Buffer := Buffer);
Pos := OPENOT_WriteSlotHeader(Offset := Pos, Key := UINT#16#0002, TypeTag := BYTE#16#03, PayloadLength := BYTE#2, Buffer := Buffer);
Pos := OPENOT_WriteU16LE(Offset := Pos, Value := Category, Buffer := Buffer);
Pos := OPENOT_WriteByte(Offset := Pos, Value := BYTE#16#00, Buffer := Buffer);
Pos := OPENOT_WriteByte(Offset := Pos, Value := BYTE#16#00, Buffer := Buffer);
Pos := OPENOT_WriteSlotHeader(Offset := Pos, Key := UINT#16#0003, TypeTag := BYTE#16#03, PayloadLength := BYTE#2, Buffer := Buffer);
Pos := OPENOT_WriteU16LE(Offset := Pos, Value := PreviousState, Buffer := Buffer);
Pos := OPENOT_WriteByte(Offset := Pos, Value := BYTE#16#00, Buffer := Buffer);
Pos := OPENOT_WriteByte(Offset := Pos, Value := BYTE#16#00, Buffer := Buffer);
Pos := OPENOT_WriteSlotHeader(Offset := Pos, Key := UINT#16#0004, TypeTag := BYTE#16#03, PayloadLength := BYTE#2, Buffer := Buffer);
Pos := OPENOT_WriteU16LE(Offset := Pos, Value := NewState, Buffer := Buffer);
Pos := OPENOT_WriteByte(Offset := Pos, Value := BYTE#16#00, Buffer := Buffer);
Pos := OPENOT_WriteByte(Offset := Pos, Value := BYTE#16#00, Buffer := Buffer);
Crc := OPENOT_Crc32c(Data := Buffer, Length := Pos);
Pos := OPENOT_WriteDWordLE(Offset := Pos, Value := Crc, Buffer := Buffer);
Length := Pos;
END_FUNCTION_BLOCK

FUNCTION_BLOCK OPENOT_EncodeCondition
VAR_INPUT
    SourceId : UDINT;
    RunId : ULINT;
    Seq : ULINT;
    SourceTime : ULINT;
    EventTypeId : UDINT;
    ConditionId : UDINT;
    ConditionClass : UINT;
    Severity : UINT;
    HasCorrelationId : BOOL;
    CorrelationId : UDINT;
    HasCauseOperand : BOOL;
    CauseOperand : UDINT;
END_VAR
VAR_OUTPUT
    Buffer : OPENOT_BYTE_BUFFER;
    Length : UINT;
END_VAR
VAR
    Pos : UINT;
    Crc : DWORD;
    TotalLength : UINT;
END_VAR

TotalLength := UINT#60;
IF HasCorrelationId THEN
    TotalLength := TotalLength + UINT#8;
END_IF;
IF EventTypeId = UDINT#16#0200 THEN
    TotalLength := TotalLength + UINT#8;
END_IF;
IF (EventTypeId = UDINT#16#0200) AND HasCauseOperand THEN
    TotalLength := TotalLength + UINT#8;
END_IF;

Pos := OPENOT_WriteHeader(
    TotalLength := TotalLength,
    Flags := UINT#16#0008,
    SourceTime := SourceTime,
    RunId := RunId,
    Seq := Seq,
    SourceId := SourceId,
    EventTypeId := EventTypeId,
    Buffer := Buffer);

Pos := OPENOT_WriteSlotHeader(Offset := Pos, Key := UINT#16#0005, TypeTag := BYTE#16#05, PayloadLength := BYTE#4, Buffer := Buffer);
Pos := OPENOT_WriteU32LE(Offset := Pos, Value := ConditionId, Buffer := Buffer);
Pos := OPENOT_WriteSlotHeader(Offset := Pos, Key := UINT#16#0006, TypeTag := BYTE#16#03, PayloadLength := BYTE#2, Buffer := Buffer);
Pos := OPENOT_WriteU16LE(Offset := Pos, Value := ConditionClass, Buffer := Buffer);
Pos := OPENOT_WriteByte(Offset := Pos, Value := BYTE#16#00, Buffer := Buffer);
Pos := OPENOT_WriteByte(Offset := Pos, Value := BYTE#16#00, Buffer := Buffer);
IF HasCorrelationId THEN
    Pos := OPENOT_WriteSlotHeader(Offset := Pos, Key := UINT#16#0007, TypeTag := BYTE#16#05, PayloadLength := BYTE#4, Buffer := Buffer);
    Pos := OPENOT_WriteU32LE(Offset := Pos, Value := CorrelationId, Buffer := Buffer);
END_IF;
IF EventTypeId = UDINT#16#0200 THEN
    Pos := OPENOT_WriteSlotHeader(Offset := Pos, Key := UINT#16#0008, TypeTag := BYTE#16#03, PayloadLength := BYTE#2, Buffer := Buffer);
    Pos := OPENOT_WriteU16LE(Offset := Pos, Value := Severity, Buffer := Buffer);
    Pos := OPENOT_WriteByte(Offset := Pos, Value := BYTE#16#00, Buffer := Buffer);
    Pos := OPENOT_WriteByte(Offset := Pos, Value := BYTE#16#00, Buffer := Buffer);
END_IF;
IF (EventTypeId = UDINT#16#0200) AND HasCauseOperand THEN
    Pos := OPENOT_WriteSlotHeader(Offset := Pos, Key := UINT#16#0009, TypeTag := BYTE#16#05, PayloadLength := BYTE#4, Buffer := Buffer);
    Pos := OPENOT_WriteU32LE(Offset := Pos, Value := CauseOperand, Buffer := Buffer);
END_IF;
Crc := OPENOT_Crc32c(Data := Buffer, Length := Pos);
Pos := OPENOT_WriteDWordLE(Offset := Pos, Value := Crc, Buffer := Buffer);
Length := Pos;
END_FUNCTION_BLOCK
